LIN {X -0.004,Y -144.888,Z 390.932,A 0.000,B 0.000,C 90.000,E1 167.757} C_DIS
LIN {X -0.050,Y -147.516,Z 390.912,A 0.000,B 0.000,C 90.000,E1 164.102} C_DIS
LIN {X 0.025,Y -150.110,Z 390.891,A 0.000,B 0.000,C 90.000,E1 160.423} C_DIS
LIN {X 0.036,Y -153.470,Z 390.871,A 0.000,B 0.000,C 90.000,E1 156.794} C_DIS
LIN {X 0.027,Y -157.832,Z 390.846,A 0.000,B 0.000,C 90.000,E1 152.308} C_DIS
LIN {X 0.058,Y -162.117,Z 390.826,A 0.000,B 0.000,C 90.000,E1 148.742} C_DIS
LIN {X -0.057,Y -166.318,Z 390.807,A 0.000,B 0.000,C 90.000,E1 145.261} C_DIS
LIN {X 0.044,Y -171.337,Z 390.788,A 0.000,B 0.000,C 90.000,E1 141.743} C_DIS
LIN {X -0.027,Y -176.238,Z 390.768,A 0.000,B 0.000,C 90.000,E1 138.324} C_DIS
LIN {X 0.092,Y -180.518,Z 390.754,A 0.000,B 0.000,C 90.000,E1 135.729} C_DIS
LIN {X 0.072,Y -185.921,Z 390.736,A 0.000,B 0.000,C 90.000,E1 132.366} C_DIS
LIN {X 0.007,Y -190.550,Z 390.722,A 0.000,B 0.000,C 90.000,E1 129.886} C_DIS
LIN {X 0.038,Y -196.301,Z 390.703,A 0.000,B 0.000,C 90.000,E1 126.583} C_DIS
LIN {X -0.023,Y -198.087,Z 390.698,A 0.000,B 0.000,C 90.000,E1 125.678} C_DIS
LIN {X -0.088,Y -297.651,Z 390.698,A 0.000,B 0.000,C 90.000,E1 125.678} C_DIS
LIN {X -0.020,Y -298.876,Z 390.698,A 0.000,B 0.000,C 90.000,E1 125.644} C_DIS
LIN {X 0.001,Y -302.899,Z 390.697,A 0.000,B 0.000,C 90.000,E1 125.471} C_DIS
LIN {X -0.050,Y -305.154,Z 390.696,A 0.000,B 0.000,C 90.000,E1 125.311} C_DIS
LIN {X 0.098,Y -308.262,Z 390.694,A 0.000,B 0.000,C 90.000,E1 124.945} C_DIS
LIN {X 0.018,Y -310.260,Z 390.693,A 0.000,B 0.000,C 90.000,E1 124.659} C_DIS
LIN {X 0.019,Y -311.830,Z 390.691,A 0.000,B 0.000,C 90.000,E1 124.358} C_DIS
LIN {X -0.017,Y -313.176,Z 390.689,A 0.000,B 0.000,C 90.000,E1 124.040} C_DIS
LIN {X 0.147,Y -324.392,Z 390.671,A 0.000,B 0.000,C 90.000,E1 120.797} C_DIS
LIN {X 0.063,Y -335.861,Z 390.655,A 0.000,B 0.000,C 90.000,E1 117.975} C_DIS
LIN {X -0.012,Y -348.771,Z 390.640,A 0.000,B 0.000,C 90.000,E1 115.207} C_DIS
LIN {X 0.098,Y -361.555,Z 390.627,A 0.000,B 0.000,C 90.000,E1 112.770} C_DIS
LIN {X -0.081,Y -375.664,Z 390.613,A 0.000,B 0.000,C 90.000,E1 110.429} C_DIS
LIN {X -0.053,Y -391.204,Z 390.601,A 0.000,B 0.000,C 90.000,E1 108.109} C_DIS
LIN {X 0.000,Y -408.288,Z 390.588,A 0.000,B 0.000,C 90.000,E1 105.843} C_DIS
LIN {X -0.024,Y -427.043,Z 390.576,A 0.000,B 0.000,C 90.000,E1 103.647} C_DIS
LIN {X 0.196,Y -447.068,Z 390.564,A 0.000,B 0.000,C 90.000,E1 101.535} C_DIS
LIN {X -0.169,Y -467.667,Z 390.554,A 0.000,B 0.000,C 90.000,E1 99.670} C_DIS
LIN {X 0.207,Y -488.731,Z 390.544,A 0.000,B 0.000,C 90.000,E1 97.871} C_DIS
LIN {X -0.132,Y -490.860,Z 390.543,A 0.000,B 0.000,C 90.000,E1 97.701} C_DIS
LIN {X -0.189,Y -492.702,Z 390.541,A 0.000,B 0.000,C 90.000,E1 97.466} C_DIS
LIN {X 0.180,Y -494.092,Z 390.540,A 0.000,B 0.000,C 90.000,E1 97.182} C_DIS
LIN {X -0.070,Y -495.891,Z 390.537,A 0.000,B 0.000,C 90.000,E1 96.720} C_DIS
LIN {X 0.180,Y -496.581,Z 390.535,A 0.000,B 0.000,C 90.000,E1 96.201} C_DIS
LIN {X -0.053,Y -496.278,Z 390.532,A 0.000,B 0.000,C 90.000,E1 95.739} C_DIS
LIN {X 0.209,Y -494.934,Z 390.529,A 0.000,B 0.000,C 90.000,E1 95.220} C_DIS
LIN {X 0.070,Y -493.801,Z 390.528,A 0.000,B 0.000,C 90.000,E1 94.992} C_DIS
LIN {X -0.026,Y -492.278,Z 390.526,A 0.000,B 0.000,C 90.000,E1 94.759} C_DIS
LIN {X -0.088,Y -484.870,Z 390.521,A 0.000,B 0.000,C 90.000,E1 93.784} C_DIS
LIN {X 0.074,Y -474.923,Z 390.514,A 0.000,B 0.000,C 90.000,E1 92.522} C_DIS
LIN {X 0.199,Y -453.804,Z 390.499,A 0.000,B 0.000,C 90.000,E1 89.714} C_DIS
LIN {X 0.116,Y -434.527,Z 390.483,A 0.000,B 0.000,C 90.000,E1 86.849} C_DIS
LIN {X 0.076,Y -415.309,Z 390.465,A 0.000,B 0.000,C 90.000,E1 83.628} C_DIS
LIN {X -0.113,Y -406.122,Z 390.456,A 0.000,B 0.000,C 90.000,E1 82.008} C_DIS
LIN {X 0.166,Y -392.691,Z 390.442,A 0.000,B 0.000,C 90.000,E1 79.454} C_DIS
LIN {X 0.149,Y -382.343,Z 390.430,A 0.000,B 0.000,C 90.000,E1 77.465} C_DIS
LIN {X 0.002,Y -370.785,Z 390.418,A 0.000,B 0.000,C 90.000,E1 75.172} C_DIS
LIN {X -0.123,Y -359.363,Z 390.405,A 0.000,B 0.000,C 90.000,E1 72.834} C_DIS
LIN {X -0.031,Y -346.929,Z 390.389,A 0.000,B 0.000,C 90.000,E1 70.115} C_DIS
LIN {X -0.056,Y -334.832,Z 390.374,A 0.000,B 0.000,C 90.000,E1 67.358} C_DIS
LIN {X 0.010,Y -320.883,Z 390.355,A 0.000,B 0.000,C 90.000,E1 63.896} C_DIS
LIN {X -0.101,Y -307.827,Z 390.335,A 0.000,B 0.000,C 90.000,E1 60.383} C_DIS
LIN {X -0.017,Y -295.740,Z 390.315,A 0.000,B 0.000,C 90.000,E1 56.755} C_DIS
LIN {X -0.058,Y -285.753,Z 390.297,A 0.000,B 0.000,C 90.000,E1 53.417} C_DIS
LIN {X 0.025,Y -278.252,Z 390.282,A 0.000,B 0.000,C 90.000,E1 50.678} C_DIS
LIN {X 0.037,Y -272.653,Z 390.270,A 0.000,B 0.000,C 90.000,E1 48.609} C_DIS
LIN {X -0.050,Y -267.017,Z 390.258,A 0.000,B 0.000,C 90.000,E1 46.539} C_DIS
LIN {X -0.068,Y -261.180,Z 390.247,A 0.000,B 0.000,C 90.000,E1 44.433} C_DIS
LIN {X -0.010,Y -255.265,Z 390.235,A 0.000,B 0.000,C 90.000,E1 42.285} C_DIS
LIN {X 0.138,Y -249.210,Z 390.223,A 0.000,B 0.000,C 90.000,E1 40.092} C_DIS
LIN {X -0.141,Y -241.139,Z 390.207,A 0.000,B 0.000,C 90.000,E1 37.237} C_DIS
LIN {X -0.052,Y -231.567,Z 390.186,A 0.000,B 0.000,C 90.000,E1 33.499} C_DIS
LIN {X 0.119,Y -222.733,Z 390.165,A 0.000,B 0.000,C 90.000,E1 29.667} C_DIS
LIN {X 0.000,Y -216.307,Z 390.148,A 0.000,B 0.000,C 90.000,E1 26.616} C_DIS
LIN {X -0.038,Y -209.169,Z 390.126,A 0.000,B 0.000,C 90.000,E1 22.717} C_DIS
LIN {X 0.047,Y -203.101,Z 390.104,A 0.000,B 0.000,C 90.000,E1 18.725} C_DIS
LIN {X 0.004,Y -197.908,Z 390.082,A 0.000,B 0.000,C 90.000,E1 14.717} C_DIS
LIN {X -0.014,Y -193.670,Z 390.059,A 0.000,B 0.000,C 90.000,E1 10.658} C_DIS
LIN {X 0.015,Y -190.579,Z 390.036,A 0.000,B 0.000,C 90.000,E1 6.549} C_DIS
LIN {X 0.086,Y -188.349,Z 390.004,A 0.000,B 0.000,C 90.000,E1 0.745} C_DIS
LIN {X 0.094,Y -189.792,Z 389.947,A 0.000,B 0.000,C 90.000,E1 350.387} C_DIS
LIN {X 0.009,Y -192.664,Z 389.919,A 0.000,B 0.000,C 90.000,E1 345.463} C_DIS
LIN {X -0.115,Y -196.117,Z 389.896,A 0.000,B 0.000,C 90.000,E1 341.402} C_DIS
LIN {X -0.005,Y -200.733,Z 389.874,A 0.000,B 0.000,C 90.000,E1 337.305} C_DIS
LIN {X 0.097,Y -206.419,Z 389.852,A 0.000,B 0.000,C 90.000,E1 333.256} C_DIS
LIN {X -0.069,Y -213.025,Z 389.830,A 0.000,B 0.000,C 90.000,E1 329.331} C_DIS
LIN {X 0.040,Y -218.897,Z 389.812,A 0.000,B 0.000,C 90.000,E1 326.167} C_DIS
LIN {X -0.010,Y -226.615,Z 389.791,A 0.000,B 0.000,C 90.000,E1 322.316} C_DIS
LIN {X -0.063,Y -235.293,Z 389.770,A 0.000,B 0.000,C 90.000,E1 318.528} C_DIS
LIN {X -0.035,Y -244.257,Z 389.751,A 0.000,B 0.000,C 90.000,E1 315.162} C_DIS
LIN {X 0.101,Y -254.424,Z 389.733,A 0.000,B 0.000,C 90.000,E1 311.838} C_DIS
LIN {X 0.056,Y -265.861,Z 389.715,A 0.000,B 0.000,C 90.000,E1 308.624} C_DIS
LIN {X 0.124,Y -276.526,Z 389.699,A 0.000,B 0.000,C 90.000,E1 305.804} C_DIS
LIN {X -0.085,Y -290.732,Z 389.680,A 0.000,B 0.000,C 90.000,E1 302.418} C_DIS
LIN {X -0.109,Y -303.015,Z 389.665,A 0.000,B 0.000,C 90.000,E1 299.745} C_DIS
LIN {X -0.141,Y -320.332,Z 389.647,A 0.000,B 0.000,C 90.000,E1 296.488} C_DIS
LIN {X -0.074,Y -331.967,Z 389.636,A 0.000,B 0.000,C 90.000,E1 294.567} C_DIS
LIN {X -0.010,Y -353.439,Z 389.619,A 0.000,B 0.000,C 90.000,E1 291.461} C_DIS
LIN {X -0.073,Y -374.118,Z 389.604,A 0.000,B 0.000,C 90.000,E1 288.779} C_DIS
LIN {X 0.168,Y -391.598,Z 389.593,A 0.000,B 0.000,C 90.000,E1 286.732} C_DIS
LIN {X 0.151,Y -412.177,Z 389.581,A 0.000,B 0.000,C 90.000,E1 284.592} C_DIS
LIN {X -0.199,Y -425.093,Z 389.574,A 0.000,B 0.000,C 90.000,E1 283.355} C_DIS
LIN {X -0.020,Y -435.184,Z 389.568,A 0.000,B 0.000,C 90.000,E1 282.299} C_DIS
LIN {X 0.211,Y -442.512,Z 389.564,A 0.000,B 0.000,C 90.000,E1 281.478} C_DIS
LIN {X 0.124,Y -449.221,Z 389.560,A 0.000,B 0.000,C 90.000,E1 280.715} C_DIS
LIN {X -0.110,Y -455.551,Z 389.555,A 0.000,B 0.000,C 90.000,E1 279.962} C_DIS
LIN {X -0.015,Y -463.211,Z 389.550,A 0.000,B 0.000,C 90.000,E1 278.916} C_DIS
LIN {X 0.172,Y -470.157,Z 389.544,A 0.000,B 0.000,C 90.000,E1 277.871} C_DIS
LIN {X -0.093,Y -476.492,Z 389.538,A 0.000,B 0.000,C 90.000,E1 276.891} C_DIS
LIN {X -0.154,Y -480.751,Z 389.534,A 0.000,B 0.000,C 90.000,E1 276.144} C_DIS
LIN {X -0.125,Y -484.413,Z 389.530,A 0.000,B 0.000,C 90.000,E1 275.391} C_DIS
LIN {X 0.181,Y -485.505,Z 389.528,A 0.000,B 0.000,C 90.000,E1 275.106} C_DIS
LIN {X -0.116,Y -487.343,Z 389.526,A 0.000,B 0.000,C 90.000,E1 274.645} C_DIS
LIN {X 0.042,Y -488.781,Z 389.523,A 0.000,B 0.000,C 90.000,E1 274.131} C_DIS
LIN {X -0.242,Y -489.894,Z 389.520,A 0.000,B 0.000,C 90.000,E1 273.669} C_DIS
LIN {X -0.060,Y -490.710,Z 389.517,A 0.000,B 0.000,C 90.000,E1 273.154} C_DIS
LIN {X 0.156,Y -491.204,Z 389.515,A 0.000,B 0.000,C 90.000,E1 272.636} C_DIS
LIN {X -0.138,Y -491.394,Z 389.512,A 0.000,B 0.000,C 90.000,E1 272.178} C_DIS
LIN {X 0.079,Y -491.252,Z 389.509,A 0.000,B 0.000,C 90.000,E1 271.661} C_DIS
LIN {X -0.210,Y -490.728,Z 389.507,A 0.000,B 0.000,C 90.000,E1 271.203} C_DIS
LIN {X -0.008,Y -489.793,Z 389.504,A 0.000,B 0.000,C 90.000,E1 270.688} C_DIS
LIN {X 0.192,Y -488.460,Z 389.501,A 0.000,B 0.000,C 90.000,E1 270.172} C_DIS
LIN {X -0.102,Y -486.512,Z 389.498,A 0.000,B 0.000,C 90.000,E1 269.714} C_DIS
LIN {X 0.083,Y -483.942,Z 389.496,A 0.000,B 0.000,C 90.000,E1 269.198} C_DIS
LIN {X -0.076,Y -482.358,Z 389.494,A 0.000,B 0.000,C 90.000,E1 268.969} C_DIS
LIN {X 0.080,Y -478.442,Z 389.491,A 0.000,B 0.000,C 90.000,E1 268.453} C_DIS
LIN {X -0.086,Y -476.104,Z 389.490,A 0.000,B 0.000,C 90.000,E1 268.224} C_DIS
LIN {X 0.228,Y -473.451,Z 389.489,A 0.000,B 0.000,C 90.000,E1 267.936} C_DIS
LIN {X 0.052,Y -470.440,Z 389.487,A 0.000,B 0.000,C 90.000,E1 267.707} C_DIS
LIN {X 0.208,Y -464.101,Z 389.485,A 0.000,B 0.000,C 90.000,E1 267.249} C_DIS
LIN {X -0.021,Y -457.142,Z 389.483,A 0.000,B 0.000,C 90.000,E1 266.906} C_DIS
LIN {X -0.093,Y -449.997,Z 389.481,A 0.000,B 0.000,C 90.000,E1 266.617} C_DIS
LIN {X -0.179,Y -442.742,Z 389.480,A 0.000,B 0.000,C 90.000,E1 266.388} C_DIS
LIN {X 0.066,Y -434.559,Z 389.479,A 0.000,B 0.000,C 90.000,E1 266.159} C_DIS
LIN {X -0.089,Y -426.538,Z 389.478,A 0.000,B 0.000,C 90.000,E1 266.045} C_DIS
LIN {X 0.188,Y -419.861,Z 389.478,A 0.000,B 0.000,C 90.000,E1 265.931} C_DIS
LIN {X -0.075,Y -408.533,Z 389.477,A 0.000,B 0.000,C 90.000,E1 265.927} C_DIS
LIN {X -0.056,Y -180.917,Z 389.477,A 0.000,B 0.000,C 90.000,E1 265.927} C_DIS
LIN {X 0.067,Y -180.868,Z 389.472,A 0.000,B 0.000,C 90.000,E1 265.008} C_DIS
LIN {X -0.056,Y -178.984,Z 389.444,A 0.000,B 0.000,C 90.000,E1 259.982} C_DIS
LIN {X -0.044,Y -177.958,Z 389.435,A 0.000,B 0.000,C 90.000,E1 258.285} C_DIS
LIN {X -0.026,Y -175.599,Z 389.411,A 0.000,B 0.000,C 90.000,E1 254.031} C_DIS
LIN {X -0.013,Y -172.323,Z 389.387,A 0.000,B 0.000,C 90.000,E1 249.752} C_DIS
LIN {X -0.034,Y -171.801,Z 389.383,A 0.000,B 0.000,C 90.000,E1 248.901} C_DIS
LIN {X 0.004,Y -169.475,Z 389.368,A 0.000,B 0.000,C 90.000,E1 246.305} C_DIS
LIN {X -0.090,Y -166.802,Z 389.349,A 0.000,B 0.000,C 90.000,E1 242.871} C_DIS
LIN {X 0.053,Y -162.783,Z 389.325,A 0.000,B 0.000,C 90.000,E1 238.456} C_DIS
LIN {X 0.029,Y -161.471,Z 389.315,A 0.000,B 0.000,C 90.000,E1 236.707} C_DIS
LIN {X 0.070,Y -157.466,Z 389.291,A 0.000,B 0.000,C 90.000,E1 232.271} C_DIS
LIN {X 0.003,Y -155.480,Z 389.276,A 0.000,B 0.000,C 90.000,E1 229.622} C_DIS
LIN {X -0.065,Y -151.789,Z 389.251,A 0.000,B 0.000,C 90.000,E1 225.162} C_DIS
LIN {X -0.051,Y -149.997,Z 389.236,A 0.000,B 0.000,C 90.000,E1 222.447} C_DIS
LIN {X -0.019,Y -146.827,Z 389.210,A 0.000,B 0.000,C 90.000,E1 217.890} C_DIS
LIN {X -0.033,Y -145.407,Z 389.195,A 0.000,B 0.000,C 90.000,E1 215.152} C_DIS
LIN {X 0.003,Y -142.838,Z 389.170,A 0.000,B 0.000,C 90.000,E1 210.541} C_DIS
LIN {X -0.067,Y -141.451,Z 389.149,A 0.000,B 0.000,C 90.000,E1 206.873} C_DIS
LIN {X -0.027,Y -139.372,Z 389.113,A 0.000,B 0.000,C 90.000,E1 200.355} C_DIS
LIN {X -0.085,Y -138.821,Z 389.098,A 0.000,B 0.000,C 90.000,E1 197.583} C_DIS
LIN {X 0.004,Y -138.353,Z 389.056,A 0.000,B 0.000,C 90.000,E1 190.074} C_DIS
LIN {X -0.023,Y -139.533,Z 389.004,A 0.000,B 0.000,C 90.000,E1 180.745} C_DIS
LIN {X 0.070,Y -141.217,Z 388.973,A 0.000,B 0.000,C 90.000,E1 175.122} C_DIS
LIN {X 0.029,Y -142.591,Z 388.958,A 0.000,B 0.000,C 90.000,E1 172.356} C_DIS
LIN {X -0.017,Y -144.892,Z 388.932,A 0.000,B 0.000,C 90.000,E1 167.757} C_DIS
LIN {X -0.064,Y -147.519,Z 388.912,A 0.000,B 0.000,C 90.000,E1 164.102} C_DIS
LIN {X 0.010,Y -150.114,Z 388.891,A 0.000,B 0.000,C 90.000,E1 160.423} C_DIS
LIN {X 0.022,Y -153.475,Z 388.871,A 0.000,B 0.000,C 90.000,E1 156.794} C_DIS
LIN {X 0.086,Y -157.838,Z 388.846,A 0.000,B 0.000,C 90.000,E1 152.281} C_DIS
LIN {X 0.043,Y -162.123,Z 388.826,A 0.000,B 0.000,C 90.000,E1 148.742} C_DIS
LIN {X -0.072,Y -166.325,Z 388.807,A 0.000,B 0.000,C 90.000,E1 145.261} C_DIS
LIN {X 0.029,Y -171.343,Z 388.788,A 0.000,B 0.000,C 90.000,E1 141.743} C_DIS
LIN {X -0.044,Y -176.245,Z 388.768,A 0.000,B 0.000,C 90.000,E1 138.324} C_DIS
LIN {X 0.076,Y -180.527,Z 388.754,A 0.000,B 0.000,C 90.000,E1 135.729} C_DIS
LIN {X 0.056,Y -185.930,Z 388.735,A 0.000,B 0.000,C 90.000,E1 132.366} C_DIS
LIN {X -0.010,Y -190.560,Z 388.722,A 0.000,B 0.000,C 90.000,E1 129.886} C_DIS
LIN {X 0.021,Y -196.310,Z 388.703,A 0.000,B 0.000,C 90.000,E1 126.583} C_DIS
LIN {X 0.084,Y -198.184,Z 388.698,A 0.000,B 0.000,C 90.000,E1 125.598} C_DIS
LIN {X 0.090,Y -297.208,Z 388.698,A 0.000,B 0.000,C 90.000,E1 125.598} C_DIS
LIN {X -0.150,Y -299.822,Z 388.698,A 0.000,B 0.000,C 90.000,E1 125.598} C_DIS
LIN {X 0.173,Y -305.154,Z 388.696,A 0.000,B 0.000,C 90.000,E1 125.231} C_DIS
LIN {X 0.073,Y -308.048,Z 388.694,A 0.000,B 0.000,C 90.000,E1 124.945} C_DIS
LIN {X -0.144,Y -310.085,Z 388.693,A 0.000,B 0.000,C 90.000,E1 124.692} C_DIS
LIN {X -0.186,Y -311.685,Z 388.691,A 0.000,B 0.000,C 90.000,E1 124.405} C_DIS
LIN {X 0.037,Y -313.091,Z 388.689,A 0.000,B 0.000,C 90.000,E1 124.040} C_DIS
LIN {X 0.010,Y -325.542,Z 388.670,A 0.000,B 0.000,C 90.000,E1 120.512} C_DIS
LIN {X -0.052,Y -337.159,Z 388.654,A 0.000,B 0.000,C 90.000,E1 117.692} C_DIS
LIN {X 0.057,Y -350.234,Z 388.638,A 0.000,B 0.000,C 90.000,E1 114.899} C_DIS
LIN {X -0.126,Y -363.174,Z 388.625,A 0.000,B 0.000,C 90.000,E1 112.514} C_DIS
LIN {X 0.075,Y -377.452,Z 388.612,A 0.000,B 0.000,C 90.000,E1 110.120} C_DIS
LIN {X 0.030,Y -393.173,Z 388.599,A 0.000,B 0.000,C 90.000,E1 107.819} C_DIS
LIN {X 0.145,Y -410.453,Z 388.587,A 0.000,B 0.000,C 90.000,E1 105.552} C_DIS
LIN {X 0.187,Y -429.421,Z 388.574,A 0.000,B 0.000,C 90.000,E1 103.355} C_DIS
LIN {X 0.143,Y -449.531,Z 388.563,A 0.000,B 0.000,C 90.000,E1 101.299} C_DIS
LIN {X -0.144,Y -470.193,Z 388.552,A 0.000,B 0.000,C 90.000,E1 99.443} C_DIS
LIN {X 0.253,Y -488.647,Z 388.544,A 0.000,B 0.000,C 90.000,E1 97.871} C_DIS
LIN {X -0.087,Y -490.843,Z 388.543,A 0.000,B 0.000,C 90.000,E1 97.701} C_DIS
LIN {X -0.106,Y -492.706,Z 388.541,A 0.000,B 0.000,C 90.000,E1 97.466} C_DIS
LIN {X -0.189,Y -494.119,Z 388.540,A 0.000,B 0.000,C 90.000,E1 97.239} C_DIS
LIN {X 0.051,Y -495.999,Z 388.537,A 0.000,B 0.000,C 90.000,E1 96.720} C_DIS
LIN {X -0.192,Y -496.756,Z 388.535,A 0.000,B 0.000,C 90.000,E1 96.258} C_DIS
LIN {X 0.068,Y -496.516,Z 388.532,A 0.000,B 0.000,C 90.000,E1 95.739} C_DIS
LIN {X -0.162,Y -495.240,Z 388.529,A 0.000,B 0.000,C 90.000,E1 95.277} C_DIS
LIN {X 0.193,Y -494.151,Z 388.528,A 0.000,B 0.000,C 90.000,E1 94.992} C_DIS
LIN {X 0.097,Y -492.683,Z 388.526,A 0.000,B 0.000,C 90.000,E1 94.759} C_DIS
LIN {X 0.038,Y -485.314,Z 388.521,A 0.000,B 0.000,C 90.000,E1 93.784} C_DIS
LIN {X 0.029,Y -473.383,Z 388.513,A 0.000,B 0.000,C 90.000,E1 92.293} C_DIS
LIN {X 0.106,Y -452.367,Z 388.497,A 0.000,B 0.000,C 90.000,E1 89.484} C_DIS
LIN {X 0.011,Y -433.226,Z 388.481,A 0.000,B 0.000,C 90.000,E1 86.617} C_DIS
LIN {X -0.052,Y -414.135,Z 388.463,A 0.000,B 0.000,C 90.000,E1 83.394} C_DIS
LIN {X -0.107,Y -401.918,Z 388.451,A 0.000,B 0.000,C 90.000,E1 81.197} C_DIS
LIN {X 0.068,Y -390.103,Z 388.439,A 0.000,B 0.000,C 90.000,E1 78.926} C_DIS
LIN {X 0.028,Y -378.336,Z 388.426,A 0.000,B 0.000,C 90.000,E1 76.645} C_DIS
LIN {X -0.098,Y -369.692,Z 388.416,A 0.000,B 0.000,C 90.000,E1 74.921} C_DIS
LIN {X 0.002,Y -358.308,Z 388.403,A 0.000,B 0.000,C 90.000,E1 72.543} C_DIS
LIN {X 0.047,Y -345.870,Z 388.388,A 0.000,B 0.000,C 90.000,E1 69.826} C_DIS
LIN {X 0.109,Y -333.768,Z 388.373,A 0.000,B 0.000,C 90.000,E1 67.050} C_DIS
LIN {X -0.104,Y -321.088,Z 388.355,A 0.000,B 0.000,C 90.000,E1 63.948} C_DIS
LIN {X 0.072,Y -308.022,Z 388.336,A 0.000,B 0.000,C 90.000,E1 60.383} C_DIS
LIN {X 0.000,Y -295.936,Z 388.315,A 0.000,B 0.000,C 90.000,E1 56.786} C_DIS
LIN {X 0.121,Y -285.921,Z 388.297,A 0.000,B 0.000,C 90.000,E1 53.417} C_DIS
LIN {X -0.013,Y -278.431,Z 388.282,A 0.000,B 0.000,C 90.000,E1 50.723} C_DIS
LIN {X 0.035,Y -272.831,Z 388.270,A 0.000,B 0.000,C 90.000,E1 48.647} C_DIS
LIN {X 0.128,Y -267.200,Z 388.259,A 0.000,B 0.000,C 90.000,E1 46.539} C_DIS
LIN {X 0.109,Y -261.392,Z 388.247,A 0.000,B 0.000,C 90.000,E1 44.433} C_DIS
LIN {X -0.005,Y -255.491,Z 388.235,A 0.000,B 0.000,C 90.000,E1 42.324} C_DIS
LIN {X -0.037,Y -249.459,Z 388.223,A 0.000,B 0.000,C 90.000,E1 40.172} C_DIS
LIN {X 0.037,Y -241.383,Z 388.207,A 0.000,B 0.000,C 90.000,E1 37.237} C_DIS
LIN {X 0.126,Y -231.829,Z 388.186,A 0.000,B 0.000,C 90.000,E1 33.499} C_DIS
LIN {X -0.006,Y -222.957,Z 388.165,A 0.000,B 0.000,C 90.000,E1 29.745} C_DIS
LIN {X -0.016,Y -216.485,Z 388.148,A 0.000,B 0.000,C 90.000,E1 26.668} C_DIS
LIN {X -0.054,Y -209.291,Z 388.126,A 0.000,B 0.000,C 90.000,E1 22.770} C_DIS
LIN {X 0.031,Y -203.189,Z 388.104,A 0.000,B 0.000,C 90.000,E1 18.779} C_DIS
LIN {X -0.014,Y -197.946,Z 388.082,A 0.000,B 0.000,C 90.000,E1 14.773} C_DIS
LIN {X -0.033,Y -193.679,Z 388.059,A 0.000,B 0.000,C 90.000,E1 10.715} C_DIS
LIN {X -0.006,Y -190.532,Z 388.037,A 0.000,B 0.000,C 90.000,E1 6.606} C_DIS
LIN {X 0.062,Y -188.290,Z 388.005,A 0.000,B 0.000,C 90.000,E1 0.802} C_DIS
LIN {X 0.089,Y -189.686,Z 387.947,A 0.000,B 0.000,C 90.000,E1 350.387} C_DIS
LIN {X -0.001,Y -192.537,Z 387.919,A 0.000,B 0.000,C 90.000,E1 345.463} C_DIS
LIN {X 0.056,Y -195.990,Z 387.896,A 0.000,B 0.000,C 90.000,E1 341.348} C_DIS
LIN {X -0.023,Y -200.597,Z 387.874,A 0.000,B 0.000,C 90.000,E1 337.305} C_DIS
LIN {X 0.074,Y -206.283,Z 387.852,A 0.000,B 0.000,C 90.000,E1 333.256} C_DIS
LIN {X -0.097,Y -212.913,Z 387.829,A 0.000,B 0.000,C 90.000,E1 329.331} C_DIS
LIN {X 0.009,Y -218.781,Z 387.812,A 0.000,B 0.000,C 90.000,E1 326.167} C_DIS
LIN {X -0.046,Y -226.510,Z 387.791,A 0.000,B 0.000,C 90.000,E1 322.316} C_DIS
LIN {X 0.073,Y -235.179,Z 387.769,A 0.000,B 0.000,C 90.000,E1 318.485} C_DIS
LIN {X -0.080,Y -244.177,Z 387.751,A 0.000,B 0.000,C 90.000,E1 315.162} C_DIS
LIN {X 0.051,Y -254.349,Z 387.732,A 0.000,B 0.000,C 90.000,E1 311.838} C_DIS
LIN {X 0.002,Y -265.796,Z 387.715,A 0.000,B 0.000,C 90.000,E1 308.624} C_DIS
LIN {X 0.066,Y -276.464,Z 387.699,A 0.000,B 0.000,C 90.000,E1 305.804} C_DIS
LIN {X -0.149,Y -290.644,Z 387.680,A 0.000,B 0.000,C 90.000,E1 302.418} C_DIS
LIN {X -0.027,Y -302.998,Z 387.665,A 0.000,B 0.000,C 90.000,E1 299.716} C_DIS
LIN {X 0.150,Y -318.508,Z 387.649,A 0.000,B 0.000,C 90.000,E1 296.744} C_DIS
LIN {X 0.155,Y -332.048,Z 387.636,A 0.000,B 0.000,C 90.000,E1 294.515} C_DIS
LIN {X -0.111,Y -351.401,Z 387.621,A 0.000,B 0.000,C 90.000,E1 291.770} C_DIS
LIN {X -0.147,Y -374.340,Z 387.604,A 0.000,B 0.000,C 90.000,E1 288.779} C_DIS
LIN {X 0.145,Y -391.804,Z 387.593,A 0.000,B 0.000,C 90.000,E1 286.732} C_DIS
LIN {X 0.146,Y -412.364,Z 387.581,A 0.000,B 0.000,C 90.000,E1 284.592} C_DIS
LIN {X 0.127,Y -425.369,Z 387.574,A 0.000,B 0.000,C 90.000,E1 283.300} C_DIS
LIN {X -0.101,Y -435.481,Z 387.568,A 0.000,B 0.000,C 90.000,E1 282.299} C_DIS
LIN {X 0.164,Y -442.670,Z 387.564,A 0.000,B 0.000,C 90.000,E1 281.478} C_DIS
LIN {X -0.048,Y -449.436,Z 387.559,A 0.000,B 0.000,C 90.000,E1 280.715} C_DIS
LIN {X 0.167,Y -455.774,Z 387.555,A 0.000,B 0.000,C 90.000,E1 279.905} C_DIS
LIN {X -0.188,Y -463.358,Z 387.549,A 0.000,B 0.000,C 90.000,E1 278.916} C_DIS
LIN {X -0.001,Y -470.282,Z 387.544,A 0.000,B 0.000,C 90.000,E1 277.871} C_DIS
LIN {X -0.122,Y -475.087,Z 387.539,A 0.000,B 0.000,C 90.000,E1 277.125} C_DIS
LIN {X 0.148,Y -480.824,Z 387.534,A 0.000,B 0.000,C 90.000,E1 276.087} C_DIS
LIN {X 0.181,Y -484.464,Z 387.530,A 0.000,B 0.000,C 90.000,E1 275.334} C_DIS
LIN {X 0.193,Y -487.339,Z 387.526,A 0.000,B 0.000,C 90.000,E1 274.588} C_DIS
LIN {X -0.135,Y -488.825,Z 387.523,A 0.000,B 0.000,C 90.000,E1 274.131} C_DIS
LIN {X 0.069,Y -489.911,Z 387.520,A 0.000,B 0.000,C 90.000,E1 273.612} C_DIS
LIN {X -0.210,Y -490.706,Z 387.517,A 0.000,B 0.000,C 90.000,E1 273.151} C_DIS
LIN {X -0.021,Y -491.180,Z 387.515,A 0.000,B 0.000,C 90.000,E1 272.636} C_DIS
LIN {X 0.176,Y -491.364,Z 387.512,A 0.000,B 0.000,C 90.000,E1 272.121} C_DIS
LIN {X -0.098,Y -491.215,Z 387.509,A 0.000,B 0.000,C 90.000,E1 271.661} C_DIS
LIN {X 0.103,Y -490.686,Z 387.506,A 0.000,B 0.000,C 90.000,E1 271.146} C_DIS
LIN {X -0.185,Y -489.748,Z 387.504,A 0.000,B 0.000,C 90.000,E1 270.688} C_DIS
LIN {X 0.015,Y -488.387,Z 387.501,A 0.000,B 0.000,C 90.000,E1 270.172} C_DIS
LIN {X 0.208,Y -486.477,Z 387.498,A 0.000,B 0.000,C 90.000,E1 269.656} C_DIS
LIN {X -0.093,Y -483.888,Z 387.495,A 0.000,B 0.000,C 90.000,E1 269.198} C_DIS
LIN {X 0.072,Y -480.390,Z 387.493,A 0.000,B 0.000,C 90.000,E1 268.682} C_DIS
LIN {X -0.095,Y -478.376,Z 387.491,A 0.000,B 0.000,C 90.000,E1 268.453} C_DIS
LIN {X 0.054,Y -473.316,Z 387.489,A 0.000,B 0.000,C 90.000,E1 267.936} C_DIS
LIN {X -0.120,Y -470.315,Z 387.487,A 0.000,B 0.000,C 90.000,E1 267.707} C_DIS
LIN {X -0.045,Y -467.301,Z 387.486,A 0.000,B 0.000,C 90.000,E1 267.478} C_DIS
LIN {X -0.056,Y -460.651,Z 387.484,A 0.000,B 0.000,C 90.000,E1 267.078} C_DIS
LIN {X 0.064,Y -453.637,Z 387.482,A 0.000,B 0.000,C 90.000,E1 266.731} C_DIS
LIN {X 0.203,Y -446.421,Z 387.480,A 0.000,B 0.000,C 90.000,E1 266.445} C_DIS
LIN {X -0.131,Y -439.021,Z 387.479,A 0.000,B 0.000,C 90.000,E1 266.274} C_DIS
LIN {X -0.071,Y -430.842,Z 387.478,A 0.000,B 0.000,C 90.000,E1 266.102} C_DIS
LIN {X 0.136,Y -419.623,Z 387.478,A 0.000,B 0.000,C 90.000,E1 265.931} C_DIS
LIN {X -0.070,Y -412.711,Z 387.477,A 0.000,B 0.000,C 90.000,E1 265.927} C_DIS
LIN {X -0.053,Y -180.917,Z 387.477,A 0.000,B 0.000,C 90.000,E1 265.927} C_DIS
LIN {X 0.049,Y -180.867,Z 387.472,A 0.000,B 0.000,C 90.000,E1 265.008} C_DIS
LIN {X -0.074,Y -178.982,Z 387.444,A 0.000,B 0.000,C 90.000,E1 259.982} C_DIS
LIN {X -0.062,Y -177.953,Z 387.435,A 0.000,B 0.000,C 90.000,E1 258.285} C_DIS
LIN {X -0.043,Y -175.595,Z 387.411,A 0.000,B 0.000,C 90.000,E1 254.031} C_DIS
LIN {X -0.030,Y -172.320,Z 387.387,A 0.000,B 0.000,C 90.000,E1 249.752} C_DIS
LIN {X -0.051,Y -171.797,Z 387.383,A 0.000,B 0.000,C 90.000,E1 248.901} C_DIS
LIN {X -0.014,Y -169.469,Z 387.368,A 0.000,B 0.000,C 90.000,E1 246.305} C_DIS
LIN {X 0.042,Y -166.797,Z 387.349,A 0.000,B 0.000,C 90.000,E1 242.820} C_DIS
LIN {X 0.036,Y -162.778,Z 387.325,A 0.000,B 0.000,C 90.000,E1 238.456} C_DIS
LIN {X 0.012,Y -161.467,Z 387.315,A 0.000,B 0.000,C 90.000,E1 236.707} C_DIS
LIN {X 0.053,Y -157.461,Z 387.290,A 0.000,B 0.000,C 90.000,E1 232.271} C_DIS
LIN {X -0.014,Y -155.473,Z 387.276,A 0.000,B 0.000,C 90.000,E1 229.622} C_DIS
LIN {X -0.081,Y -151.784,Z 387.251,A 0.000,B 0.000,C 90.000,E1 225.162} C_DIS
LIN {X -0.068,Y -149.992,Z 387.236,A 0.000,B 0.000,C 90.000,E1 222.447} C_DIS
LIN {X -0.035,Y -146.823,Z 387.210,A 0.000,B 0.000,C 90.000,E1 217.890} C_DIS
LIN {X 0.070,Y -145.402,Z 387.195,A 0.000,B 0.000,C 90.000,E1 215.105} C_DIS
LIN {X -0.013,Y -142.835,Z 387.170,A 0.000,B 0.000,C 90.000,E1 210.541} C_DIS
LIN {X 0.044,Y -141.448,Z 387.149,A 0.000,B 0.000,C 90.000,E1 206.821} C_DIS
LIN {X -0.043,Y -139.371,Z 387.113,A 0.000,B 0.000,C 90.000,E1 200.355} C_DIS
LIN {X 0.032,Y -138.819,Z 387.097,A 0.000,B 0.000,C 90.000,E1 197.528} C_DIS
LIN {X -0.012,Y -138.352,Z 387.056,A 0.000,B 0.000,C 90.000,E1 190.074} C_DIS
LIN {X -0.039,Y -139.534,Z 387.004,A 0.000,B 0.000,C 90.000,E1 180.745} C_DIS
LIN {X 0.054,Y -141.220,Z 386.973,A 0.000,B 0.000,C 90.000,E1 175.122} C_DIS
LIN {X 0.013,Y -142.593,Z 386.958,A 0.000,B 0.000,C 90.000,E1 172.356} C_DIS
LIN {X -0.034,Y -144.895,Z 386.932,A 0.000,B 0.000,C 90.000,E1 167.757} C_DIS
LIN {X -0.080,Y -147.524,Z 386.911,A 0.000,B 0.000,C 90.000,E1 164.102} C_DIS
LIN {X -0.006,Y -150.120,Z 386.891,A 0.000,B 0.000,C 90.000,E1 160.423} C_DIS
LIN {X 0.005,Y -153.482,Z 386.871,A 0.000,B 0.000,C 90.000,E1 156.794} C_DIS
LIN {X 0.069,Y -157.845,Z 386.846,A 0.000,B 0.000,C 90.000,E1 152.281} C_DIS
LIN {X 0.025,Y -162.131,Z 386.826,A 0.000,B 0.000,C 90.000,E1 148.742} C_DIS
LIN {X 0.005,Y -166.333,Z 386.807,A 0.000,B 0.000,C 90.000,E1 145.229} C_DIS
LIN {X 0.011,Y -171.351,Z 386.787,A 0.000,B 0.000,C 90.000,E1 141.743} C_DIS
LIN {X -0.062,Y -176.255,Z 386.768,A 0.000,B 0.000,C 90.000,E1 138.324} C_DIS
LIN {X 0.057,Y -180.538,Z 386.754,A 0.000,B 0.000,C 90.000,E1 135.729} C_DIS
LIN {X 0.037,Y -185.939,Z 386.735,A 0.000,B 0.000,C 90.000,E1 132.366} C_DIS
LIN {X -0.029,Y -190.570,Z 386.722,A 0.000,B 0.000,C 90.000,E1 129.886} C_DIS
LIN {X 0.002,Y -196.320,Z 386.703,A 0.000,B 0.000,C 90.000,E1 126.583} C_DIS
LIN {X -0.086,Y -198.281,Z 386.698,A 0.000,B 0.000,C 90.000,E1 125.598} C_DIS
LIN {X -0.180,Y -297.492,Z 386.698,A 0.000,B 0.000,C 90.000,E1 125.598} C_DIS
LIN {X 0.102,Y -302.486,Z 386.697,A 0.000,B 0.000,C 90.000,E1 125.391} C_DIS
LIN {X 0.142,Y -304.752,Z 386.696,A 0.000,B 0.000,C 90.000,E1 125.231} C_DIS
LIN {X 0.042,Y -307.824,Z 386.694,A 0.000,B 0.000,C 90.000,E1 124.945} C_DIS
LIN {X -0.073,Y -311.471,Z 386.691,A 0.000,B 0.000,C 90.000,E1 124.405} C_DIS
LIN {X -0.033,Y -312.959,Z 386.689,A 0.000,B 0.000,C 90.000,E1 124.072} C_DIS
LIN {X -0.055,Y -325.454,Z 386.670,A 0.000,B 0.000,C 90.000,E1 120.541} C_DIS
LIN {X -0.109,Y -337.061,Z 386.654,A 0.000,B 0.000,C 90.000,E1 117.719} C_DIS
LIN {X 0.158,Y -350.128,Z 386.638,A 0.000,B 0.000,C 90.000,E1 114.899} C_DIS
LIN {X -0.024,Y -363.058,Z 386.625,A 0.000,B 0.000,C 90.000,E1 112.514} C_DIS
LIN {X 0.178,Y -377.326,Z 386.612,A 0.000,B 0.000,C 90.000,E1 110.120} C_DIS
LIN {X 0.135,Y -393.037,Z 386.599,A 0.000,B 0.000,C 90.000,E1 107.819} C_DIS
LIN {X -0.144,Y -410.306,Z 386.587,A 0.000,B 0.000,C 90.000,E1 105.607} C_DIS
LIN {X -0.124,Y -429.262,Z 386.574,A 0.000,B 0.000,C 90.000,E1 103.411} C_DIS
LIN {X 0.245,Y -449.367,Z 386.563,A 0.000,B 0.000,C 90.000,E1 101.299} C_DIS
LIN {X -0.047,Y -470.025,Z 386.552,A 0.000,B 0.000,C 90.000,E1 99.443} C_DIS
LIN {X -0.205,Y -488.485,Z 386.544,A 0.000,B 0.000,C 90.000,E1 97.936} C_DIS
LIN {X 0.006,Y -490.774,Z 386.543,A 0.000,B 0.000,C 90.000,E1 97.701} C_DIS
LIN {X 0.036,Y -492.661,Z 386.542,A 0.000,B 0.000,C 90.000,E1 97.466} C_DIS
LIN {X 0.002,Y -494.100,Z 386.540,A 0.000,B 0.000,C 90.000,E1 97.239} C_DIS
LIN {X -0.250,Y -496.084,Z 386.537,A 0.000,B 0.000,C 90.000,E1 96.777} C_DIS
LIN {X 0.000,Y -496.923,Z 386.535,A 0.000,B 0.000,C 90.000,E1 96.258} C_DIS
LIN {X -0.233,Y -496.758,Z 386.532,A 0.000,B 0.000,C 90.000,E1 95.796} C_DIS
LIN {X 0.031,Y -495.569,Z 386.529,A 0.000,B 0.000,C 90.000,E1 95.277} C_DIS
LIN {X -0.106,Y -494.531,Z 386.528,A 0.000,B 0.000,C 90.000,E1 95.049} C_DIS
LIN {X -0.200,Y -493.127,Z 386.527,A 0.000,B 0.000,C 90.000,E1 94.816} C_DIS
LIN {X -0.139,Y -487.701,Z 386.523,A 0.000,B 0.000,C 90.000,E1 94.073} C_DIS
LIN {X -0.214,Y -479.903,Z 386.517,A 0.000,B 0.000,C 90.000,E1 93.094} C_DIS
LIN {X 0.087,Y -454.686,Z 386.499,A 0.000,B 0.000,C 90.000,E1 89.771} C_DIS
LIN {X 0.036,Y -435.315,Z 386.483,A 0.000,B 0.000,C 90.000,E1 86.906} C_DIS
LIN {X 0.027,Y -416.034,Z 386.465,A 0.000,B 0.000,C 90.000,E1 83.685} C_DIS
LIN {X -0.093,Y -405.337,Z 386.454,A 0.000,B 0.000,C 90.000,E1 81.781} C_DIS
LIN {X 0.224,Y -391.988,Z 386.440,A 0.000,B 0.000,C 90.000,E1 79.218} C_DIS
LIN {X 0.197,Y -381.653,Z 386.429,A 0.000,B 0.000,C 90.000,E1 77.229} C_DIS
LIN {X 0.034,Y -371.547,Z 386.418,A 0.000,B 0.000,C 90.000,E1 75.227} C_DIS
LIN {X -0.177,Y -360.109,Z 386.405,A 0.000,B 0.000,C 90.000,E1 72.906} C_DIS
LIN {X -0.108,Y -348.952,Z 386.392,A 0.000,B 0.000,C 90.000,E1 70.496} C_DIS
LIN {X 0.043,Y -338.068,Z 386.378,A 0.000,B 0.000,C 90.000,E1 68.028} C_DIS
LIN {X -0.012,Y -325.069,Z 386.361,A 0.000,B 0.000,C 90.000,E1 64.921} C_DIS
LIN {X 0.141,Y -311.710,Z 386.341,A 0.000,B 0.000,C 90.000,E1 61.385} C_DIS
LIN {X 0.150,Y -300.413,Z 386.323,A 0.000,B 0.000,C 90.000,E1 58.122} C_DIS
LIN {X 0.083,Y -290.048,Z 386.305,A 0.000,B 0.000,C 90.000,E1 54.815} C_DIS
LIN {X -0.030,Y -280.480,Z 386.286,A 0.000,B 0.000,C 90.000,E1 51.457} C_DIS
LIN {X 0.061,Y -274.933,Z 386.274,A 0.000,B 0.000,C 90.000,E1 49.380} C_DIS
LIN {X -0.023,Y -267.417,Z 386.259,A 0.000,B 0.000,C 90.000,E1 46.620} C_DIS
LIN {X -0.035,Y -261.634,Z 386.247,A 0.000,B 0.000,C 90.000,E1 44.514} C_DIS
LIN {X 0.031,Y -255.757,Z 386.235,A 0.000,B 0.000,C 90.000,E1 42.366} C_DIS
LIN {X -0.004,Y -249.736,Z 386.223,A 0.000,B 0.000,C 90.000,E1 40.216} C_DIS
LIN {X -0.078,Y -241.644,Z 386.207,A 0.000,B 0.000,C 90.000,E1 37.317} C_DIS
LIN {X 0.027,Y -232.104,Z 386.187,A 0.000,B 0.000,C 90.000,E1 33.579} C_DIS
LIN {X 0.023,Y -223.211,Z 386.166,A 0.000,B 0.000,C 90.000,E1 29.795} C_DIS
LIN {X -0.084,Y -216.688,Z 386.148,A 0.000,B 0.000,C 90.000,E1 26.744} C_DIS
LIN {X -0.026,Y -209.433,Z 386.127,A 0.000,B 0.000,C 90.000,E1 22.823} C_DIS
LIN {X -0.009,Y -203.295,Z 386.105,A 0.000,B 0.000,C 90.000,E1 18.852} C_DIS
LIN {X 0.011,Y -198.005,Z 386.082,A 0.000,B 0.000,C 90.000,E1 14.828} C_DIS
LIN {X -0.046,Y -193.703,Z 386.060,A 0.000,B 0.000,C 90.000,E1 10.782} C_DIS
LIN {X 0.015,Y -190.523,Z 386.037,A 0.000,B 0.000,C 90.000,E1 6.663} C_DIS
LIN {X 0.081,Y -188.245,Z 386.005,A 0.000,B 0.000,C 90.000,E1 0.859} C_DIS
LIN {X 0.084,Y -189.578,Z 385.947,A 0.000,B 0.000,C 90.000,E1 350.387} C_DIS
LIN {X -0.009,Y -192.409,Z 385.919,A 0.000,B 0.000,C 90.000,E1 345.463} C_DIS
LIN {X 0.044,Y -195.869,Z 385.896,A 0.000,B 0.000,C 90.000,E1 341.348} C_DIS
LIN {X 0.037,Y -200.458,Z 385.874,A 0.000,B 0.000,C 90.000,E1 337.283} C_DIS
LIN {X 0.053,Y -206.173,Z 385.852,A 0.000,B 0.000,C 90.000,E1 333.256} C_DIS
LIN {X 0.060,Y -212.818,Z 385.829,A 0.000,B 0.000,C 90.000,E1 329.282} C_DIS
LIN {X -0.021,Y -218.652,Z 385.812,A 0.000,B 0.000,C 90.000,E1 326.167} C_DIS
LIN {X 0.099,Y -226.408,Z 385.791,A 0.000,B 0.000,C 90.000,E1 322.271} C_DIS
LIN {X 0.033,Y -235.070,Z 385.769,A 0.000,B 0.000,C 90.000,E1 318.485} C_DIS
LIN {X -0.123,Y -244.100,Z 385.751,A 0.000,B 0.000,C 90.000,E1 315.162} C_DIS
LIN {X 0.004,Y -254.271,Z 385.732,A 0.000,B 0.000,C 90.000,E1 311.838} C_DIS
LIN {X -0.049,Y -265.719,Z 385.715,A 0.000,B 0.000,C 90.000,E1 308.624} C_DIS
LIN {X 0.010,Y -276.396,Z 385.699,A 0.000,B 0.000,C 90.000,E1 305.804} C_DIS
LIN {X 0.191,Y -290.567,Z 385.680,A 0.000,B 0.000,C 90.000,E1 302.339} C_DIS
LIN {X 0.171,Y -302.975,Z 385.665,A 0.000,B 0.000,C 90.000,E1 299.667} C_DIS
LIN {X 0.081,Y -318.541,Z 385.649,A 0.000,B 0.000,C 90.000,E1 296.744} C_DIS
LIN {X -0.017,Y -330.117,Z 385.638,A 0.000,B 0.000,C 90.000,E1 294.847} C_DIS
LIN {X 0.128,Y -349.373,Z 385.622,A 0.000,B 0.000,C 90.000,E1 292.025} C_DIS
LIN {X 0.088,Y -369.782,Z 385.607,A 0.000,B 0.000,C 90.000,E1 289.322} C_DIS
LIN {X 0.108,Y -387.058,Z 385.596,A 0.000,B 0.000,C 90.000,E1 287.275} C_DIS
LIN {X -0.149,Y -407.642,Z 385.584,A 0.000,B 0.000,C 90.000,E1 285.134} C_DIS
LIN {X 0.030,Y -423.300,Z 385.575,A 0.000,B 0.000,C 90.000,E1 283.536} C_DIS
LIN {X -0.198,Y -433.472,Z 385.569,A 0.000,B 0.000,C 90.000,E1 282.535} C_DIS
LIN {X 0.041,Y -440.802,Z 385.565,A 0.000,B 0.000,C 90.000,E1 281.715} C_DIS
LIN {X -0.179,Y -447.695,Z 385.561,A 0.000,B 0.000,C 90.000,E1 280.950} C_DIS
LIN {X -0.179,Y -456.112,Z 385.555,A 0.000,B 0.000,C 90.000,E1 279.905} C_DIS
LIN {X 0.096,Y -461.845,Z 385.551,A 0.000,B 0.000,C 90.000,E1 279.095} C_DIS
LIN {X -0.192,Y -468.873,Z 385.545,A 0.000,B 0.000,C 90.000,E1 278.106} C_DIS
LIN {X -0.001,Y -475.303,Z 385.539,A 0.000,B 0.000,C 90.000,E1 277.068} C_DIS
LIN {X -0.203,Y -481.005,Z 385.534,A 0.000,B 0.000,C 90.000,E1 276.087} C_DIS
LIN {X -0.172,Y -484.618,Z 385.530,A 0.000,B 0.000,C 90.000,E1 275.334} C_DIS
LIN {X -0.160,Y -487.442,Z 385.525,A 0.000,B 0.000,C 90.000,E1 274.588} C_DIS
LIN {X -0.001,Y -488.873,Z 385.523,A 0.000,B 0.000,C 90.000,E1 274.073} C_DIS
LIN {X 0.205,Y -489.942,Z 385.520,A 0.000,B 0.000,C 90.000,E1 273.555} C_DIS
LIN {X -0.075,Y -490.716,Z 385.517,A 0.000,B 0.000,C 90.000,E1 273.094} C_DIS
LIN {X 0.114,Y -491.177,Z 385.514,A 0.000,B 0.000,C 90.000,E1 272.579} C_DIS
LIN {X -0.179,Y -491.319,Z 385.512,A 0.000,B 0.000,C 90.000,E1 272.121} C_DIS
LIN {X 0.038,Y -491.130,Z 385.509,A 0.000,B 0.000,C 90.000,E1 271.604} C_DIS
LIN {X 0.239,Y -490.597,Z 385.506,A 0.000,B 0.000,C 90.000,E1 271.088} C_DIS
LIN {X -0.049,Y -489.654,Z 385.503,A 0.000,B 0.000,C 90.000,E1 270.630} C_DIS
LIN {X 0.149,Y -488.258,Z 385.501,A 0.000,B 0.000,C 90.000,E1 270.115} C_DIS
LIN {X -0.145,Y -486.264,Z 385.498,A 0.000,B 0.000,C 90.000,E1 269.656} C_DIS
LIN {X 0.039,Y -483.683,Z 385.495,A 0.000,B 0.000,C 90.000,E1 269.141} C_DIS
LIN {X 0.201,Y -480.192,Z 385.492,A 0.000,B 0.000,C 90.000,E1 268.625} C_DIS
LIN {X -0.118,Y -475.695,Z 385.490,A 0.000,B 0.000,C 90.000,E1 268.165} C_DIS
LIN {X 0.181,Y -472.997,Z 385.488,A 0.000,B 0.000,C 90.000,E1 267.879} C_DIS
LIN {X 0.004,Y -469.921,Z 385.487,A 0.000,B 0.000,C 90.000,E1 267.650} C_DIS
LIN {X 0.107,Y -466.938,Z 385.486,A 0.000,B 0.000,C 90.000,E1 267.421} C_DIS
LIN {X 0.160,Y -460.245,Z 385.484,A 0.000,B 0.000,C 90.000,E1 267.020} C_DIS
LIN {X 0.111,Y -456.725,Z 385.483,A 0.000,B 0.000,C 90.000,E1 266.849} C_DIS
LIN {X 0.032,Y -449.289,Z 385.481,A 0.000,B 0.000,C 90.000,E1 266.560} C_DIS
LIN {X -0.011,Y -441.961,Z 385.480,A 0.000,B 0.000,C 90.000,E1 266.331} C_DIS
LIN {X -0.104,Y -434.172,Z 385.479,A 0.000,B 0.000,C 90.000,E1 266.159} C_DIS
LIN {X 0.174,Y -425.900,Z 385.478,A 0.000,B 0.000,C 90.000,E1 265.988} C_DIS
LIN {X 0.068,Y -418.557,Z 385.477,A 0.000,B 0.000,C 90.000,E1 265.927} C_DIS
LIN {X -0.114,Y -412.308,Z 385.477,A 0.000,B 0.000,C 90.000,E1 265.927} C_DIS
LIN {X -0.071,Y -180.916,Z 385.477,A 0.000,B 0.000,C 90.000,E1 265.927} C_DIS
LIN {X 0.023,Y -180.865,Z 385.472,A 0.000,B 0.000,C 90.000,E1 265.008} C_DIS
LIN {X 0.075,Y -178.979,Z 385.444,A 0.000,B 0.000,C 90.000,E1 259.926} C_DIS
LIN {X 0.085,Y -177.948,Z 385.435,A 0.000,B 0.000,C 90.000,E1 258.229} C_DIS
LIN {X -0.069,Y -175.589,Z 385.411,A 0.000,B 0.000,C 90.000,E1 254.031} C_DIS
LIN {X -0.056,Y -172.314,Z 385.387,A 0.000,B 0.000,C 90.000,E1 249.752} C_DIS
LIN {X -0.077,Y -171.792,Z 385.383,A 0.000,B 0.000,C 90.000,E1 248.901} C_DIS
LIN {X -0.039,Y -169.462,Z 385.368,A 0.000,B 0.000,C 90.000,E1 246.305} C_DIS
LIN {X 0.016,Y -166.791,Z 385.349,A 0.000,B 0.000,C 90.000,E1 242.820} C_DIS
LIN {X 0.012,Y -162.770,Z 385.325,A 0.000,B 0.000,C 90.000,E1 238.456} C_DIS
LIN {X -0.012,Y -161.460,Z 385.315,A 0.000,B 0.000,C 90.000,E1 236.707} C_DIS
LIN {X 0.029,Y -157.454,Z 385.290,A 0.000,B 0.000,C 90.000,E1 232.271} C_DIS
LIN {X -0.038,Y -155.465,Z 385.276,A 0.000,B 0.000,C 90.000,E1 229.622} C_DIS
LIN {X 0.003,Y -151.779,Z 385.251,A 0.000,B 0.000,C 90.000,E1 225.121} C_DIS
LIN {X 0.020,Y -149.985,Z 385.236,A 0.000,B 0.000,C 90.000,E1 222.405} C_DIS
LIN {X -0.059,Y -146.817,Z 385.210,A 0.000,B 0.000,C 90.000,E1 217.890} C_DIS
LIN {X 0.047,Y -145.396,Z 385.195,A 0.000,B 0.000,C 90.000,E1 215.105} C_DIS
LIN {X -0.035,Y -142.831,Z 385.170,A 0.000,B 0.000,C 90.000,E1 210.541} C_DIS
LIN {X 0.021,Y -141.444,Z 385.149,A 0.000,B 0.000,C 90.000,E1 206.821} C_DIS
LIN {X 0.065,Y -139.369,Z 385.113,A 0.000,B 0.000,C 90.000,E1 200.301} C_DIS
LIN {X 0.051,Y -138.817,Z 385.097,A 0.000,B 0.000,C 90.000,E1 197.511} C_DIS
LIN {X -0.034,Y -138.352,Z 385.056,A 0.000,B 0.000,C 90.000,E1 190.074} C_DIS
LIN {X -0.061,Y -139.536,Z 385.004,A 0.000,B 0.000,C 90.000,E1 180.745} C_DIS
LIN {X 0.032,Y -141.225,Z 384.973,A 0.000,B 0.000,C 90.000,E1 175.122} C_DIS
LIN {X -0.010,Y -142.596,Z 384.958,A 0.000,B 0.000,C 90.000,E1 172.356} C_DIS
LIN {X -0.056,Y -144.901,Z 384.932,A 0.000,B 0.000,C 90.000,E1 167.757} C_DIS
LIN {X 0.038,Y -147.529,Z 384.911,A 0.000,B 0.000,C 90.000,E1 164.047} C_DIS
LIN {X -0.030,Y -150.127,Z 384.891,A 0.000,B 0.000,C 90.000,E1 160.423} C_DIS
LIN {X -0.018,Y -153.491,Z 384.871,A 0.000,B 0.000,C 90.000,E1 156.794} C_DIS
LIN {X 0.045,Y -157.855,Z 384.846,A 0.000,B 0.000,C 90.000,E1 152.281} C_DIS
LIN {X 0.001,Y -162.141,Z 384.826,A 0.000,B 0.000,C 90.000,E1 148.742} C_DIS
LIN {X -0.021,Y -166.345,Z 384.807,A 0.000,B 0.000,C 90.000,E1 145.229} C_DIS
LIN {X -0.015,Y -171.362,Z 384.787,A 0.000,B 0.000,C 90.000,E1 141.743} C_DIS
LIN {X -0.087,Y -176.268,Z 384.768,A 0.000,B 0.000,C 90.000,E1 138.324} C_DIS
LIN {X 0.031,Y -180.552,Z 384.754,A 0.000,B 0.000,C 90.000,E1 135.729} C_DIS
LIN {X 0.010,Y -185.954,Z 384.735,A 0.000,B 0.000,C 90.000,E1 132.366} C_DIS
LIN {X 0.066,Y -190.586,Z 384.721,A 0.000,B 0.000,C 90.000,E1 129.850} C_DIS
LIN {X -0.027,Y -196.335,Z 384.703,A 0.000,B 0.000,C 90.000,E1 126.583} C_DIS
LIN {X 0.000,Y -198.390,Z 384.697,A 0.000,B 0.000,C 90.000,E1 125.518} C_DIS
LIN {X -0.049,Y -298.045,Z 384.697,A 0.000,B 0.000,C 90.000,E1 125.518} C_DIS
LIN {X -0.149,Y -299.228,Z 384.697,A 0.000,B 0.000,C 90.000,E1 125.518} C_DIS
LIN {X -0.076,Y -304.767,Z 384.696,A 0.000,B 0.000,C 90.000,E1 125.231} C_DIS
LIN {X -0.001,Y -307.604,Z 384.694,A 0.000,B 0.000,C 90.000,E1 124.945} C_DIS
LIN {X -0.036,Y -311.313,Z 384.691,A 0.000,B 0.000,C 90.000,E1 124.405} C_DIS
LIN {X 0.003,Y -312.866,Z 384.689,A 0.000,B 0.000,C 90.000,E1 124.072} C_DIS
LIN {X 0.070,Y -316.228,Z 384.684,A 0.000,B 0.000,C 90.000,E1 123.086} C_DIS
LIN {X 0.078,Y -326.629,Z 384.668,A 0.000,B 0.000,C 90.000,E1 120.207} C_DIS
LIN {X 0.055,Y -338.392,Z 384.652,A 0.000,B 0.000,C 90.000,E1 117.385} C_DIS
LIN {X -0.101,Y -351.620,Z 384.637,A 0.000,B 0.000,C 90.000,E1 114.643} C_DIS
LIN {X 0.079,Y -364.709,Z 384.623,A 0.000,B 0.000,C 90.000,E1 112.206} C_DIS
LIN {X -0.029,Y -379.147,Z 384.610,A 0.000,B 0.000,C 90.000,E1 109.866} C_DIS
LIN {X -0.163,Y -395.042,Z 384.598,A 0.000,B 0.000,C 90.000,E1 107.583} C_DIS
LIN {X -0.005,Y -412.510,Z 384.585,A 0.000,B 0.000,C 90.000,E1 105.315} C_DIS
LIN {X 0.100,Y -431.658,Z 384.573,A 0.000,B 0.000,C 90.000,E1 103.119} C_DIS
LIN {X 0.124,Y -451.835,Z 384.562,A 0.000,B 0.000,C 90.000,E1 101.074} C_DIS
LIN {X 0.077,Y -472.556,Z 384.551,A 0.000,B 0.000,C 90.000,E1 99.208} C_DIS
LIN {X -0.176,Y -488.412,Z 384.544,A 0.000,B 0.000,C 90.000,E1 97.936} C_DIS
LIN {X 0.034,Y -490.765,Z 384.543,A 0.000,B 0.000,C 90.000,E1 97.701} C_DIS
LIN {X 0.034,Y -492.671,Z 384.542,A 0.000,B 0.000,C 90.000,E1 97.473} C_DIS
LIN {X 0.099,Y -494.126,Z 384.540,A 0.000,B 0.000,C 90.000,E1 97.239} C_DIS
LIN {X 0.005,Y -495.316,Z 384.539,A 0.000,B 0.000,C 90.000,E1 97.004} C_DIS
LIN {X -0.152,Y -496.180,Z 384.538,A 0.000,B 0.000,C 90.000,E1 96.777} C_DIS
LIN {X 0.105,Y -497.072,Z 384.535,A 0.000,B 0.000,C 90.000,E1 96.258} C_DIS
LIN {X -0.128,Y -496.967,Z 384.532,A 0.000,B 0.000,C 90.000,E1 95.796} C_DIS
LIN {X 0.137,Y -495.840,Z 384.529,A 0.000,B 0.000,C 90.000,E1 95.277} C_DIS
LIN {X 0.000,Y -494.841,Z 384.528,A 0.000,B 0.000,C 90.000,E1 95.049} C_DIS
LIN {X -0.135,Y -493.483,Z 384.527,A 0.000,B 0.000,C 90.000,E1 94.821} C_DIS
LIN {X -0.031,Y -488.133,Z 384.523,A 0.000,B 0.000,C 90.000,E1 94.073} C_DIS
LIN {X 0.212,Y -478.339,Z 384.516,A 0.000,B 0.000,C 90.000,E1 92.808} C_DIS
LIN {X -0.019,Y -453.217,Z 384.497,A 0.000,B 0.000,C 90.000,E1 89.542} C_DIS
LIN {X -0.083,Y -433.993,Z 384.481,A 0.000,B 0.000,C 90.000,E1 86.674} C_DIS
LIN {X -0.115,Y -414.828,Z 384.464,A 0.000,B 0.000,C 90.000,E1 83.451} C_DIS
LIN {X -0.150,Y -402.673,Z 384.451,A 0.000,B 0.000,C 90.000,E1 81.254} C_DIS
LIN {X -0.027,Y -390.865,Z 384.439,A 0.000,B 0.000,C 90.000,E1 78.993} C_DIS
LIN {X -0.001,Y -380.553,Z 384.428,A 0.000,B 0.000,C 90.000,E1 76.992} C_DIS
LIN {X -0.088,Y -369.010,Z 384.415,A 0.000,B 0.000,C 90.000,E1 74.685} C_DIS
LIN {X -0.009,Y -357.617,Z 384.402,A 0.000,B 0.000,C 90.000,E1 72.308} C_DIS
LIN {X 0.108,Y -346.511,Z 384.388,A 0.000,B 0.000,C 90.000,E1 69.880} C_DIS
LIN {X 0.191,Y -334.318,Z 384.373,A 0.000,B 0.000,C 90.000,E1 67.102} C_DIS
LIN {X -0.144,Y -321.541,Z 384.356,A 0.000,B 0.000,C 90.000,E1 64.024} C_DIS
LIN {X 0.042,Y -308.457,Z 384.336,A 0.000,B 0.000,C 90.000,E1 60.461} C_DIS
LIN {X 0.140,Y -296.361,Z 384.316,A 0.000,B 0.000,C 90.000,E1 56.834} C_DIS
LIN {X 0.109,Y -286.294,Z 384.297,A 0.000,B 0.000,C 90.000,E1 53.497} C_DIS
LIN {X -0.018,Y -278.807,Z 384.282,A 0.000,B 0.000,C 90.000,E1 50.803} C_DIS
LIN {X 0.037,Y -273.235,Z 384.271,A 0.000,B 0.000,C 90.000,E1 48.728} C_DIS
LIN {X -0.058,Y -267.598,Z 384.259,A 0.000,B 0.000,C 90.000,E1 46.662} C_DIS
LIN {X 0.125,Y -261.846,Z 384.247,A 0.000,B 0.000,C 90.000,E1 44.514} C_DIS
LIN {X 0.018,Y -255.983,Z 384.236,A 0.000,B 0.000,C 90.000,E1 42.405} C_DIS
LIN {X -0.004,Y -249.971,Z 384.224,A 0.000,B 0.000,C 90.000,E1 40.253} C_DIS
LIN {X 0.083,Y -241.884,Z 384.207,A 0.000,B 0.000,C 90.000,E1 37.317} C_DIS
LIN {X -0.129,Y -234.197,Z 384.191,A 0.000,B 0.000,C 90.000,E1 34.405} C_DIS
LIN {X 0.056,Y -225.145,Z 384.170,A 0.000,B 0.000,C 90.000,E1 30.590} C_DIS
LIN {X 0.098,Y -218.422,Z 384.153,A 0.000,B 0.000,C 90.000,E1 27.513} C_DIS
LIN {X 0.014,Y -210.946,Z 384.131,A 0.000,B 0.000,C 90.000,E1 23.643} C_DIS
LIN {X 0.019,Y -205.733,Z 384.114,A 0.000,B 0.000,C 90.000,E1 20.482} C_DIS
LIN {X -0.021,Y -200.076,Z 384.092,A 0.000,B 0.000,C 90.000,E1 16.496} C_DIS
LIN {X 0.115,Y -195.357,Z 384.069,A 0.000,B 0.000,C 90.000,E1 12.411} C_DIS
LIN {X 0.058,Y -191.628,Z 384.046,A 0.000,B 0.000,C 90.000,E1 8.341} C_DIS
LIN {X -0.090,Y -188.872,Z 384.019,A 0.000,B 0.000,C 90.000,E1 3.440} C_DIS
LIN {X 0.021,Y -189.846,Z 383.942,A 0.000,B 0.000,C 90.000,E1 349.577} C_DIS
LIN {X 0.021,Y -192.917,Z 383.915,A 0.000,B 0.000,C 90.000,E1 344.629} C_DIS
LIN {X -0.034,Y -196.586,Z 383.892,A 0.000,B 0.000,C 90.000,E1 340.550} C_DIS
LIN {X -0.018,Y -201.405,Z 383.869,A 0.000,B 0.000,C 90.000,E1 336.485} C_DIS
LIN {X 0.032,Y -206.061,Z 383.851,A 0.000,B 0.000,C 90.000,E1 333.256} C_DIS
LIN {X 0.036,Y -212.725,Z 383.829,A 0.000,B 0.000,C 90.000,E1 329.282} C_DIS
LIN {X -0.048,Y -218.521,Z 383.812,A 0.000,B 0.000,C 90.000,E1 326.167} C_DIS
LIN {X 0.067,Y -226.305,Z 383.790,A 0.000,B 0.000,C 90.000,E1 322.271} C_DIS
LIN {X -0.002,Y -234.980,Z 383.769,A 0.000,B 0.000,C 90.000,E1 318.485} C_DIS
LIN {X 0.009,Y -244.025,Z 383.751,A 0.000,B 0.000,C 90.000,E1 315.121} C_DIS
LIN {X -0.054,Y -253.007,Z 383.734,A 0.000,B 0.000,C 90.000,E1 312.204} C_DIS
LIN {X 0.012,Y -264.328,Z 383.716,A 0.000,B 0.000,C 90.000,E1 308.955} C_DIS
LIN {X 0.028,Y -274.982,Z 383.701,A 0.000,B 0.000,C 90.000,E1 306.137} C_DIS
LIN {X 0.000,Y -289.012,Z 383.682,A 0.000,B 0.000,C 90.000,E1 302.704} C_DIS
LIN {X 0.094,Y -301.327,Z 383.667,A 0.000,B 0.000,C 90.000,E1 300.001} C_DIS
LIN {X -0.041,Y -316.741,Z 383.650,A 0.000,B 0.000,C 90.000,E1 297.078} C_DIS
LIN {X 0.057,Y -330.237,Z 383.638,A 0.000,B 0.000,C 90.000,E1 294.823} C_DIS
LIN {X 0.061,Y -349.574,Z 383.622,A 0.000,B 0.000,C 90.000,E1 292.025} C_DIS
LIN {X -0.012,Y -372.379,Z 383.606,A 0.000,B 0.000,C 90.000,E1 289.033} C_DIS
LIN {X 0.108,Y -389.885,Z 383.594,A 0.000,B 0.000,C 90.000,E1 286.985} C_DIS
LIN {X 0.123,Y -408.156,Z 383.584,A 0.000,B 0.000,C 90.000,E1 285.064} C_DIS
LIN {X 0.169,Y -423.822,Z 383.575,A 0.000,B 0.000,C 90.000,E1 283.480} C_DIS
LIN {X -0.064,Y -433.954,Z 383.569,A 0.000,B 0.000,C 90.000,E1 282.479} C_DIS
LIN {X 0.169,Y -441.229,Z 383.565,A 0.000,B 0.000,C 90.000,E1 281.658} C_DIS
LIN {X -0.045,Y -448.081,Z 383.560,A 0.000,B 0.000,C 90.000,E1 280.894} C_DIS
LIN {X -0.037,Y -456.400,Z 383.555,A 0.000,B 0.000,C 90.000,E1 279.849} C_DIS
LIN {X -0.139,Y -462.126,Z 383.550,A 0.000,B 0.000,C 90.000,E1 279.086} C_DIS
LIN {X -0.194,Y -470.760,Z 383.543,A 0.000,B 0.000,C 90.000,E1 277.814} C_DIS
LIN {X 0.017,Y -476.983,Z 383.538,A 0.000,B 0.000,C 90.000,E1 276.777} C_DIS
LIN {X -0.037,Y -481.147,Z 383.533,A 0.000,B 0.000,C 90.000,E1 276.030} C_DIS
LIN {X -0.003,Y -484.714,Z 383.529,A 0.000,B 0.000,C 90.000,E1 275.277} C_DIS
LIN {X 0.012,Y -487.483,Z 383.525,A 0.000,B 0.000,C 90.000,E1 274.531} C_DIS
LIN {X 0.207,Y -488.902,Z 383.522,A 0.000,B 0.000,C 90.000,E1 274.012} C_DIS
LIN {X -0.111,Y -489.957,Z 383.520,A 0.000,B 0.000,C 90.000,E1 273.555} C_DIS
LIN {X 0.100,Y -490.700,Z 383.517,A 0.000,B 0.000,C 90.000,E1 273.037} C_DIS
LIN {X -0.201,Y -491.131,Z 383.514,A 0.000,B 0.000,C 90.000,E1 272.579} C_DIS
LIN {X -0.004,Y -491.292,Z 383.511,A 0.000,B 0.000,C 90.000,E1 272.064} C_DIS
LIN {X 0.213,Y -491.085,Z 383.509,A 0.000,B 0.000,C 90.000,E1 271.547} C_DIS
LIN {X -0.077,Y -490.541,Z 383.506,A 0.000,B 0.000,C 90.000,E1 271.088} C_DIS
LIN {X 0.125,Y -489.573,Z 383.503,A 0.000,B 0.000,C 90.000,E1 270.573} C_DIS
LIN {X -0.165,Y -488.162,Z 383.501,A 0.000,B 0.000,C 90.000,E1 270.115} C_DIS
LIN {X -0.124,Y -484.889,Z 383.496,A 0.000,B 0.000,C 90.000,E1 269.370} C_DIS
LIN {X 0.210,Y -483.491,Z 383.495,A 0.000,B 0.000,C 90.000,E1 269.083} C_DIS
LIN {X -0.110,Y -479.970,Z 383.492,A 0.000,B 0.000,C 90.000,E1 268.625} C_DIS
LIN {X 0.048,Y -475.422,Z 383.490,A 0.000,B 0.000,C 90.000,E1 268.108} C_DIS
LIN {X -0.128,Y -472.669,Z 383.488,A 0.000,B 0.000,C 90.000,E1 267.879} C_DIS
LIN {X 0.166,Y -469.567,Z 383.487,A 0.000,B 0.000,C 90.000,E1 267.593} C_DIS
LIN {X -0.189,Y -466.529,Z 383.486,A 0.000,B 0.000,C 90.000,E1 267.421} C_DIS
LIN {X -0.113,Y -459.817,Z 383.483,A 0.000,B 0.000,C 90.000,E1 267.020} C_DIS
LIN {X 0.110,Y -452.834,Z 383.482,A 0.000,B 0.000,C 90.000,E1 266.674} C_DIS
LIN {X -0.123,Y -445.700,Z 383.480,A 0.000,B 0.000,C 90.000,E1 266.445} C_DIS
LIN {X 0.044,Y -438.146,Z 383.479,A 0.000,B 0.000,C 90.000,E1 266.216} C_DIS
LIN {X 0.142,Y -430.029,Z 383.478,A 0.000,B 0.000,C 90.000,E1 266.045} C_DIS
LIN {X 0.151,Y -420.831,Z 383.478,A 0.000,B 0.000,C 90.000,E1 265.931} C_DIS
LIN {X -0.148,Y -412.157,Z 383.477,A 0.000,B 0.000,C 90.000,E1 265.927} C_DIS
LIN {X 0.094,Y -180.916,Z 383.477,A 0.000,B 0.000,C 90.000,E1 265.869} C_DIS
LIN {X -0.043,Y -180.830,Z 383.472,A 0.000,B 0.000,C 90.000,E1 264.894} C_DIS
LIN {X 0.031,Y -178.867,Z 383.442,A 0.000,B 0.000,C 90.000,E1 259.634} C_DIS
LIN {X -0.068,Y -175.909,Z 383.414,A 0.000,B 0.000,C 90.000,E1 254.574} C_DIS
LIN {X -0.011,Y -174.597,Z 383.405,A 0.000,B 0.000,C 90.000,E1 252.851} C_DIS
LIN {X -0.085,Y -171.579,Z 383.381,A 0.000,B 0.000,C 90.000,E1 248.592} C_DIS
LIN {X -0.095,Y -167.802,Z 383.357,A 0.000,B 0.000,C 90.000,E1 244.280} C_DIS
LIN {X 0.070,Y -166.520,Z 383.347,A 0.000,B 0.000,C 90.000,E1 242.487} C_DIS
LIN {X 0.059,Y -162.521,Z 383.323,A 0.000,B 0.000,C 90.000,E1 238.122} C_DIS
LIN {X 0.030,Y -161.194,Z 383.313,A 0.000,B 0.000,C 90.000,E1 236.373} C_DIS
LIN {X -0.068,Y -157.204,Z 383.289,A 0.000,B 0.000,C 90.000,E1 231.984} C_DIS
LIN {X -0.045,Y -155.933,Z 383.279,A 0.000,B 0.000,C 90.000,E1 230.194} C_DIS
LIN {X -0.085,Y -152.184,Z 383.254,A 0.000,B 0.000,C 90.000,E1 225.729} C_DIS
LIN {X -0.064,Y -150.431,Z 383.239,A 0.000,B 0.000,C 90.000,E1 223.014} C_DIS
LIN {X -0.036,Y -147.159,Z 383.214,A 0.000,B 0.000,C 90.000,E1 218.463} C_DIS
LIN {X -0.068,Y -145.173,Z 383.193,A 0.000,B 0.000,C 90.000,E1 214.818} C_DIS
LIN {X -0.032,Y -142.323,Z 383.163,A 0.000,B 0.000,C 90.000,E1 209.283} C_DIS
LIN {X -0.038,Y -141.712,Z 383.152,A 0.000,B 0.000,C 90.000,E1 207.436} C_DIS
LIN {X 0.010,Y -139.472,Z 383.116,A 0.000,B 0.000,C 90.000,E1 200.918} C_DIS
LIN {X -0.068,Y -139.204,Z 383.106,A 0.000,B 0.000,C 90.000,E1 199.087} C_DIS
LIN {X -0.010,Y -138.330,Z 383.054,A 0.000,B 0.000,C 90.000,E1 189.726} C_DIS
LIN {X -0.007,Y -139.439,Z 383.007,A 0.000,B 0.000,C 90.000,E1 181.318} C_DIS
LIN {X -0.067,Y -140.971,Z 382.976,A 0.000,B 0.000,C 90.000,E1 175.755} C_DIS
LIN {X 0.024,Y -142.727,Z 382.956,A 0.000,B 0.000,C 90.000,E1 172.008} C_DIS
LIN {X -0.019,Y -145.112,Z 382.930,A 0.000,B 0.000,C 90.000,E1 167.409} C_DIS
LIN {X -0.024,Y -147.735,Z 382.910,A 0.000,B 0.000,C 90.000,E1 163.740} C_DIS
LIN {X 0.058,Y -150.399,Z 382.889,A 0.000,B 0.000,C 90.000,E1 160.061} C_DIS
LIN {X -0.067,Y -153.834,Z 382.869,A 0.000,B 0.000,C 90.000,E1 156.485} C_DIS
LIN {X -0.008,Y -157.245,Z 382.849,A 0.000,B 0.000,C 90.000,E1 152.871} C_DIS
LIN {X -0.068,Y -161.417,Z 382.829,A 0.000,B 0.000,C 90.000,E1 149.331} C_DIS
LIN {X -0.059,Y -165.619,Z 382.810,A 0.000,B 0.000,C 90.000,E1 145.801} C_DIS
LIN {X 0.061,Y -170.547,Z 382.790,A 0.000,B 0.000,C 90.000,E1 142.271} C_DIS
LIN {X -0.031,Y -175.426,Z 382.771,A 0.000,B 0.000,C 90.000,E1 138.852} C_DIS
LIN {X 0.086,Y -181.049,Z 382.752,A 0.000,B 0.000,C 90.000,E1 135.405} C_DIS
LIN {X -0.047,Y -186.484,Z 382.734,A 0.000,B 0.000,C 90.000,E1 132.081} C_DIS
LIN {X 0.020,Y -191.105,Z 382.720,A 0.000,B 0.000,C 90.000,E1 129.564} C_DIS
LIN {X -0.059,Y -196.899,Z 382.702,A 0.000,B 0.000,C 90.000,E1 126.297} C_DIS
LIN {X -0.024,Y -198.498,Z 382.697,A 0.000,B 0.000,C 90.000,E1 125.471} C_DIS
LIN {X 0.100,Y -298.212,Z 382.697,A 0.000,B 0.000,C 90.000,E1 125.438} C_DIS
LIN {X 0.021,Y -300.873,Z 382.697,A 0.000,B 0.000,C 90.000,E1 125.391} C_DIS
LIN {X -0.010,Y -306.537,Z 382.695,A 0.000,B 0.000,C 90.000,E1 125.025} C_DIS
LIN {X -0.043,Y -309.621,Z 382.693,A 0.000,B 0.000,C 90.000,E1 124.659} C_DIS
LIN {X 0.008,Y -311.567,Z 382.691,A 0.000,B 0.000,C 90.000,E1 124.326} C_DIS
LIN {X 0.062,Y -313.086,Z 382.689,A 0.000,B 0.000,C 90.000,E1 123.992} C_DIS
LIN {X -0.165,Y -318.636,Z 382.680,A 0.000,B 0.000,C 90.000,E1 122.418} C_DIS
LIN {X -0.095,Y -329.363,Z 382.664,A 0.000,B 0.000,C 90.000,E1 119.539} C_DIS
LIN {X 0.101,Y -341.473,Z 382.648,A 0.000,B 0.000,C 90.000,E1 116.693} C_DIS
LIN {X 0.004,Y -353.490,Z 382.635,A 0.000,B 0.000,C 90.000,E1 114.259} C_DIS
LIN {X 0.095,Y -366.776,Z 382.621,A 0.000,B 0.000,C 90.000,E1 111.844} C_DIS
LIN {X 0.043,Y -381.426,Z 382.608,A 0.000,B 0.000,C 90.000,E1 109.504} C_DIS
LIN {X -0.030,Y -397.551,Z 382.596,A 0.000,B 0.000,C 90.000,E1 107.221} C_DIS
LIN {X 0.197,Y -415.268,Z 382.583,A 0.000,B 0.000,C 90.000,E1 104.954} C_DIS
LIN {X -0.116,Y -434.644,Z 382.571,A 0.000,B 0.000,C 90.000,E1 102.827} C_DIS
LIN {X 0.113,Y -454.908,Z 382.560,A 0.000,B 0.000,C 90.000,E1 100.782} C_DIS
LIN {X -0.208,Y -475.706,Z 382.550,A 0.000,B 0.000,C 90.000,E1 98.973} C_DIS
LIN {X -0.014,Y -488.958,Z 382.544,A 0.000,B 0.000,C 90.000,E1 97.871} C_DIS
LIN {X 0.130,Y -491.218,Z 382.543,A 0.000,B 0.000,C 90.000,E1 97.644} C_DIS
LIN {X -0.147,Y -492.938,Z 382.541,A 0.000,B 0.000,C 90.000,E1 97.466} C_DIS
LIN {X 0.181,Y -494.478,Z 382.540,A 0.000,B 0.000,C 90.000,E1 97.182} C_DIS
LIN {X 0.082,Y -495.629,Z 382.539,A 0.000,B 0.000,C 90.000,E1 96.947} C_DIS
LIN {X -0.161,Y -497.001,Z 382.536,A 0.000,B 0.000,C 90.000,E1 96.486} C_DIS
LIN {X 0.096,Y -497.329,Z 382.533,A 0.000,B 0.000,C 90.000,E1 95.967} C_DIS
LIN {X -0.182,Y -496.661,Z 382.530,A 0.000,B 0.000,C 90.000,E1 95.511} C_DIS
LIN {X 0.085,Y -494.887,Z 382.528,A 0.000,B 0.000,C 90.000,E1 94.992} C_DIS
LIN {X -0.009,Y -493.478,Z 382.526,A 0.000,B 0.000,C 90.000,E1 94.759} C_DIS
LIN {X 0.094,Y -488.098,Z 382.522,A 0.000,B 0.000,C 90.000,E1 94.012} C_DIS
LIN {X -0.183,Y -478.287,Z 382.515,A 0.000,B 0.000,C 90.000,E1 92.808} C_DIS
LIN {X 0.063,Y -453.161,Z 382.497,A 0.000,B 0.000,C 90.000,E1 89.484} C_DIS
LIN {X -0.195,Y -435.597,Z 382.483,A 0.000,B 0.000,C 90.000,E1 86.906} C_DIS
LIN {X -0.183,Y -416.308,Z 382.465,A 0.000,B 0.000,C 90.000,E1 83.685} C_DIS
LIN {X -0.189,Y -404.160,Z 382.453,A 0.000,B 0.000,C 90.000,E1 81.489} C_DIS
LIN {X 0.039,Y -392.319,Z 382.440,A 0.000,B 0.000,C 90.000,E1 79.218} C_DIS
LIN {X 0.020,Y -382.025,Z 382.429,A 0.000,B 0.000,C 90.000,E1 77.229} C_DIS
LIN {X -0.131,Y -370.447,Z 382.416,A 0.000,B 0.000,C 90.000,E1 74.936} C_DIS
LIN {X 0.081,Y -359.017,Z 382.403,A 0.000,B 0.000,C 90.000,E1 72.543} C_DIS
LIN {X 0.116,Y -347.840,Z 382.390,A 0.000,B 0.000,C 90.000,E1 70.134} C_DIS
LIN {X -0.083,Y -336.915,Z 382.376,A 0.000,B 0.000,C 90.000,E1 67.720} C_DIS
LIN {X -0.032,Y -323.963,Z 382.359,A 0.000,B 0.000,C 90.000,E1 64.588} C_DIS
LIN {X 0.092,Y -310.697,Z 382.339,A 0.000,B 0.000,C 90.000,E1 61.051} C_DIS
LIN {X 0.073,Y -299.473,Z 382.321,A 0.000,B 0.000,C 90.000,E1 57.788} C_DIS
LIN {X -0.024,Y -289.170,Z 382.303,A 0.000,B 0.000,C 90.000,E1 54.482} C_DIS
LIN {X 0.006,Y -279.675,Z 382.284,A 0.000,B 0.000,C 90.000,E1 51.090} C_DIS
LIN {X 0.079,Y -274.145,Z 382.272,A 0.000,B 0.000,C 90.000,E1 49.013} C_DIS
LIN {X 0.016,Y -268.510,Z 382.261,A 0.000,B 0.000,C 90.000,E1 46.944} C_DIS
LIN {X 0.022,Y -262.763,Z 382.249,A 0.000,B 0.000,C 90.000,E1 44.838} C_DIS
LIN {X 0.110,Y -256.969,Z 382.237,A 0.000,B 0.000,C 90.000,E1 42.690} C_DIS
LIN {X 0.100,Y -250.971,Z 382.225,A 0.000,B 0.000,C 90.000,E1 40.539} C_DIS
LIN {X 0.013,Y -242.875,Z 382.209,A 0.000,B 0.000,C 90.000,E1 37.649} C_DIS
LIN {X 0.015,Y -235.154,Z 382.193,A 0.000,B 0.000,C 90.000,E1 34.692} C_DIS
LIN {X 0.035,Y -226.025,Z 382.172,A 0.000,B 0.000,C 90.000,E1 30.924} C_DIS
LIN {X -0.093,Y -219.213,Z 382.155,A 0.000,B 0.000,C 90.000,E1 27.897} C_DIS
LIN {X -0.061,Y -211.619,Z 382.133,A 0.000,B 0.000,C 90.000,E1 24.003} C_DIS
LIN {X -0.041,Y -206.297,Z 382.116,A 0.000,B 0.000,C 90.000,E1 20.844} C_DIS
LIN {X -0.064,Y -200.531,Z 382.094,A 0.000,B 0.000,C 90.000,E1 16.858} C_DIS
LIN {X -0.098,Y -195.705,Z 382.071,A 0.000,B 0.000,C 90.000,E1 12.827} C_DIS
LIN {X -0.104,Y -191.857,Z 382.048,A 0.000,B 0.000,C 90.000,E1 8.746} C_DIS
LIN {X -0.037,Y -188.984,Z 382.021,A 0.000,B 0.000,C 90.000,E1 3.784} C_DIS
LIN {X -0.006,Y -190.154,Z 381.938,A 0.000,B 0.000,C 90.000,E1 348.757} C_DIS
LIN {X 0.057,Y -193.467,Z 381.910,A 0.000,B 0.000,C 90.000,E1 343.795} C_DIS
LIN {X 0.079,Y -197.360,Z 381.887,A 0.000,B 0.000,C 90.000,E1 339.699} C_DIS
LIN {X 0.014,Y -202.411,Z 381.865,A 0.000,B 0.000,C 90.000,E1 335.665} C_DIS
LIN {X -0.097,Y -207.245,Z 381.847,A 0.000,B 0.000,C 90.000,E1 332.487} C_DIS
LIN {X 0.042,Y -214.058,Z 381.825,A 0.000,B 0.000,C 90.000,E1 328.486} C_DIS
LIN {X -0.060,Y -221.420,Z 381.803,A 0.000,B 0.000,C 90.000,E1 324.609} C_DIS
LIN {X -0.091,Y -227.905,Z 381.786,A 0.000,B 0.000,C 90.000,E1 321.537} C_DIS
LIN {X -0.036,Y -234.903,Z 381.769,A 0.000,B 0.000,C 90.000,E1 318.485} C_DIS
LIN {X -0.027,Y -243.946,Z 381.751,A 0.000,B 0.000,C 90.000,E1 315.121} C_DIS
LIN {X 0.080,Y -251.755,Z 381.736,A 0.000,B 0.000,C 90.000,E1 312.528} C_DIS
LIN {X 0.125,Y -262.992,Z 381.718,A 0.000,B 0.000,C 90.000,E1 309.277} C_DIS
LIN {X -0.100,Y -273.580,Z 381.703,A 0.000,B 0.000,C 90.000,E1 306.503} C_DIS
LIN {X -0.019,Y -287.449,Z 381.684,A 0.000,B 0.000,C 90.000,E1 303.038} C_DIS
LIN {X 0.038,Y -301.296,Z 381.667,A 0.000,B 0.000,C 90.000,E1 300.001} C_DIS
LIN {X -0.011,Y -314.974,Z 381.652,A 0.000,B 0.000,C 90.000,E1 297.385} C_DIS
LIN {X -0.040,Y -326.334,Z 381.641,A 0.000,B 0.000,C 90.000,E1 295.463} C_DIS
LIN {X -0.106,Y -336.673,Z 381.633,A 0.000,B 0.000,C 90.000,E1 293.898} C_DIS
LIN {X 0.050,Y -354.229,Z 381.619,A 0.000,B 0.000,C 90.000,E1 291.408} C_DIS
LIN {X -0.069,Y -372.597,Z 381.606,A 0.000,B 0.000,C 90.000,E1 289.033} C_DIS
LIN {X -0.129,Y -389.912,Z 381.595,A 0.000,B 0.000,C 90.000,E1 287.040} C_DIS
LIN {X -0.109,Y -407.988,Z 381.584,A 0.000,B 0.000,C 90.000,E1 285.134} C_DIS
LIN {X 0.075,Y -423.549,Z 381.575,A 0.000,B 0.000,C 90.000,E1 283.536} C_DIS
LIN {X -0.198,Y -433.719,Z 381.569,A 0.000,B 0.000,C 90.000,E1 282.535} C_DIS
LIN {X 0.013,Y -441.010,Z 381.565,A 0.000,B 0.000,C 90.000,E1 281.715} C_DIS
LIN {X 0.021,Y -449.982,Z 381.559,A 0.000,B 0.000,C 90.000,E1 280.658} C_DIS
LIN {X 0.052,Y -458.125,Z 381.553,A 0.000,B 0.000,C 90.000,E1 279.613} C_DIS
LIN {X -0.104,Y -463.678,Z 381.549,A 0.000,B 0.000,C 90.000,E1 278.859} C_DIS
LIN {X 0.089,Y -470.501,Z 381.543,A 0.000,B 0.000,C 90.000,E1 277.814} C_DIS
LIN {X -0.172,Y -476.745,Z 381.538,A 0.000,B 0.000,C 90.000,E1 276.834} C_DIS
LIN {X 0.113,Y -482.222,Z 381.532,A 0.000,B 0.000,C 90.000,E1 275.796} C_DIS
LIN {X 0.107,Y -485.531,Z 381.528,A 0.000,B 0.000,C 90.000,E1 275.049} C_DIS
LIN {X -0.190,Y -487.312,Z 381.525,A 0.000,B 0.000,C 90.000,E1 274.588} C_DIS
LIN {X -0.032,Y -488.757,Z 381.523,A 0.000,B 0.000,C 90.000,E1 274.073} C_DIS
LIN {X 0.173,Y -489.826,Z 381.520,A 0.000,B 0.000,C 90.000,E1 273.555} C_DIS
LIN {X -0.108,Y -490.606,Z 381.517,A 0.000,B 0.000,C 90.000,E1 273.094} C_DIS
LIN {X 0.082,Y -491.059,Z 381.514,A 0.000,B 0.000,C 90.000,E1 272.579} C_DIS
LIN {X -0.212,Y -491.244,Z 381.512,A 0.000,B 0.000,C 90.000,E1 272.121} C_DIS
LIN {X 0.003,Y -491.076,Z 381.509,A 0.000,B 0.000,C 90.000,E1 271.604} C_DIS
LIN {X 0.204,Y -490.550,Z 381.506,A 0.000,B 0.000,C 90.000,E1 271.088} C_DIS
LIN {X -0.084,Y -489.598,Z 381.503,A 0.000,B 0.000,C 90.000,E1 270.630} C_DIS
LIN {X 0.114,Y -488.202,Z 381.501,A 0.000,B 0.000,C 90.000,E1 270.115} C_DIS
LIN {X -0.180,Y -486.275,Z 381.498,A 0.000,B 0.000,C 90.000,E1 269.656} C_DIS
LIN {X 0.155,Y -485.088,Z 381.497,A 0.000,B 0.000,C 90.000,E1 269.370} C_DIS
LIN {X -0.155,Y -482.116,Z 381.494,A 0.000,B 0.000,C 90.000,E1 268.912} C_DIS
LIN {X -0.001,Y -478.196,Z 381.491,A 0.000,B 0.000,C 90.000,E1 268.396} C_DIS
LIN {X 0.146,Y -473.156,Z 381.488,A 0.000,B 0.000,C 90.000,E1 267.879} C_DIS
LIN {X -0.029,Y -470.132,Z 381.487,A 0.000,B 0.000,C 90.000,E1 267.650} C_DIS
LIN {X 0.054,Y -467.103,Z 381.486,A 0.000,B 0.000,C 90.000,E1 267.421} C_DIS
LIN {X 0.077,Y -460.452,Z 381.483,A 0.000,B 0.000,C 90.000,E1 267.020} C_DIS
LIN {X -0.210,Y -453.462,Z 381.482,A 0.000,B 0.000,C 90.000,E1 266.731} C_DIS
LIN {X -0.052,Y -446.261,Z 381.480,A 0.000,B 0.000,C 90.000,E1 266.445} C_DIS
LIN {X 0.061,Y -438.588,Z 381.479,A 0.000,B 0.000,C 90.000,E1 266.216} C_DIS
LIN {X 0.125,Y -430.245,Z 381.478,A 0.000,B 0.000,C 90.000,E1 266.045} C_DIS
LIN {X 0.126,Y -420.934,Z 381.477,A 0.000,B 0.000,C 90.000,E1 265.931} C_DIS
LIN {X -0.179,Y -411.735,Z 381.477,A 0.000,B 0.000,C 90.000,E1 265.927} C_DIS
LIN {X 0.081,Y -180.916,Z 381.477,A 0.000,B 0.000,C 90.000,E1 265.869} C_DIS
LIN {X -0.057,Y -180.829,Z 381.472,A 0.000,B 0.000,C 90.000,E1 264.894} C_DIS
LIN {X 0.017,Y -178.864,Z 381.442,A 0.000,B 0.000,C 90.000,E1 259.634} C_DIS
LIN {X -0.082,Y -175.908,Z 381.414,A 0.000,B 0.000,C 90.000,E1 254.574} C_DIS
LIN {X 0.026,Y -174.593,Z 381.405,A 0.000,B 0.000,C 90.000,E1 252.834} C_DIS
LIN {X 0.061,Y -171.575,Z 381.381,A 0.000,B 0.000,C 90.000,E1 248.539} C_DIS
LIN {X 0.043,Y -167.798,Z 381.357,A 0.000,B 0.000,C 90.000,E1 244.229} C_DIS
LIN {X 0.057,Y -166.515,Z 381.347,A 0.000,B 0.000,C 90.000,E1 242.487} C_DIS
LIN {X 0.052,Y -163.223,Z 381.328,A 0.000,B 0.000,C 90.000,E1 238.997} C_DIS
LIN {X 0.017,Y -161.189,Z 381.313,A 0.000,B 0.000,C 90.000,E1 236.373} C_DIS
LIN {X -0.081,Y -157.201,Z 381.289,A 0.000,B 0.000,C 90.000,E1 231.984} C_DIS
LIN {X -0.058,Y -155.929,Z 381.279,A 0.000,B 0.000,C 90.000,E1 230.194} C_DIS
LIN {X 0.012,Y -152.181,Z 381.254,A 0.000,B 0.000,C 90.000,E1 225.688} C_DIS
LIN {X 0.027,Y -150.428,Z 381.239,A 0.000,B 0.000,C 90.000,E1 222.975} C_DIS
LIN {X -0.048,Y -147.155,Z 381.214,A 0.000,B 0.000,C 90.000,E1 218.463} C_DIS
LIN {X -0.080,Y -145.171,Z 381.193,A 0.000,B 0.000,C 90.000,E1 214.818} C_DIS
LIN {X -0.045,Y -142.320,Z 381.163,A 0.000,B 0.000,C 90.000,E1 209.283} C_DIS
LIN {X 0.075,Y -141.710,Z 381.152,A 0.000,B 0.000,C 90.000,E1 207.385} C_DIS
LIN {X -0.002,Y -139.471,Z 381.116,A 0.000,B 0.000,C 90.000,E1 200.918} C_DIS
LIN {X 0.052,Y -139.203,Z 381.106,A 0.000,B 0.000,C 90.000,E1 199.033} C_DIS
LIN {X -0.022,Y -138.328,Z 381.054,A 0.000,B 0.000,C 90.000,E1 189.726} C_DIS
LIN {X -0.019,Y -139.439,Z 381.007,A 0.000,B 0.000,C 90.000,E1 181.318} C_DIS
LIN {X 0.061,Y -140.973,Z 380.976,A 0.000,B 0.000,C 90.000,E1 175.698} C_DIS
LIN {X 0.011,Y -142.729,Z 380.956,A 0.000,B 0.000,C 90.000,E1 172.008} C_DIS
LIN {X -0.031,Y -145.115,Z 380.930,A 0.000,B 0.000,C 90.000,E1 167.409} C_DIS
LIN {X -0.037,Y -147.739,Z 380.910,A 0.000,B 0.000,C 90.000,E1 163.740} C_DIS
LIN {X 0.045,Y -150.403,Z 380.889,A 0.000,B 0.000,C 90.000,E1 160.061} C_DIS
LIN {X -0.081,Y -153.839,Z 380.869,A 0.000,B 0.000,C 90.000,E1 156.485} C_DIS
LIN {X -0.022,Y -157.250,Z 380.849,A 0.000,B 0.000,C 90.000,E1 152.871} C_DIS
LIN {X 0.057,Y -161.423,Z 380.829,A 0.000,B 0.000,C 90.000,E1 149.282} C_DIS
LIN {X -0.073,Y -165.625,Z 380.810,A 0.000,B 0.000,C 90.000,E1 145.801} C_DIS
LIN {X 0.047,Y -170.554,Z 380.790,A 0.000,B 0.000,C 90.000,E1 142.271} C_DIS
LIN {X -0.045,Y -175.433,Z 380.771,A 0.000,B 0.000,C 90.000,E1 138.852} C_DIS
LIN {X 0.072,Y -181.055,Z 380.752,A 0.000,B 0.000,C 90.000,E1 135.405} C_DIS
LIN {X -0.062,Y -186.492,Z 380.734,A 0.000,B 0.000,C 90.000,E1 132.081} C_DIS
LIN {X 0.005,Y -191.113,Z 380.720,A 0.000,B 0.000,C 90.000,E1 129.564} C_DIS
LIN {X -0.074,Y -196.907,Z 380.702,A 0.000,B 0.000,C 90.000,E1 126.297} C_DIS
LIN {X -0.055,Y -198.582,Z 380.697,A 0.000,B 0.000,C 90.000,E1 125.438} C_DIS
LIN {X 0.106,Y -297.659,Z 380.697,A 0.000,B 0.000,C 90.000,E1 125.391} C_DIS
LIN {X -0.003,Y -299.371,Z 380.697,A 0.000,B 0.000,C 90.000,E1 125.391} C_DIS
LIN {X 0.107,Y -303.804,Z 380.696,A 0.000,B 0.000,C 90.000,E1 125.185} C_DIS
LIN {X -0.033,Y -306.193,Z 380.695,A 0.000,B 0.000,C 90.000,E1 125.025} C_DIS
LIN {X -0.067,Y -309.441,Z 380.692,A 0.000,B 0.000,C 90.000,E1 124.659} C_DIS
LIN {X 0.048,Y -311.398,Z 380.691,A 0.000,B 0.000,C 90.000,E1 124.326} C_DIS
LIN {X -0.093,Y -312.934,Z 380.689,A 0.000,B 0.000,C 90.000,E1 124.040} C_DIS
LIN {X 0.010,Y -315.269,Z 380.685,A 0.000,B 0.000,C 90.000,E1 123.372} C_DIS
LIN {X 0.158,Y -325.545,Z 380.669,A 0.000,B 0.000,C 90.000,E1 120.463} C_DIS
LIN {X 0.105,Y -337.175,Z 380.654,A 0.000,B 0.000,C 90.000,E1 117.641} C_DIS
LIN {X -0.085,Y -350.259,Z 380.638,A 0.000,B 0.000,C 90.000,E1 114.899} C_DIS
LIN {X 0.064,Y -363.210,Z 380.625,A 0.000,B 0.000,C 90.000,E1 112.461} C_DIS
LIN {X -0.076,Y -377.500,Z 380.612,A 0.000,B 0.000,C 90.000,E1 110.120} C_DIS
LIN {X -0.125,Y -393.234,Z 380.599,A 0.000,B 0.000,C 90.000,E1 107.819} C_DIS
LIN {X -0.014,Y -410.528,Z 380.586,A 0.000,B 0.000,C 90.000,E1 105.552} C_DIS
LIN {X 0.028,Y -429.504,Z 380.574,A 0.000,B 0.000,C 90.000,E1 103.355} C_DIS
LIN {X -0.014,Y -449.620,Z 380.563,A 0.000,B 0.000,C 90.000,E1 101.299} C_DIS
LIN {X 0.243,Y -470.287,Z 380.552,A 0.000,B 0.000,C 90.000,E1 99.378} C_DIS
LIN {X 0.082,Y -488.783,Z 380.544,A 0.000,B 0.000,C 90.000,E1 97.871} C_DIS
LIN {X -0.238,Y -491.114,Z 380.543,A 0.000,B 0.000,C 90.000,E1 97.701} C_DIS
LIN {X -0.007,Y -492.884,Z 380.541,A 0.000,B 0.000,C 90.000,E1 97.466} C_DIS
LIN {X -0.169,Y -494.486,Z 380.540,A 0.000,B 0.000,C 90.000,E1 97.239} C_DIS
LIN {X 0.222,Y -495.686,Z 380.539,A 0.000,B 0.000,C 90.000,E1 96.947} C_DIS
LIN {X -0.020,Y -497.136,Z 380.536,A 0.000,B 0.000,C 90.000,E1 96.486} C_DIS
LIN {X 0.237,Y -497.530,Z 380.533,A 0.000,B 0.000,C 90.000,E1 95.967} C_DIS
LIN {X -0.041,Y -496.931,Z 380.531,A 0.000,B 0.000,C 90.000,E1 95.511} C_DIS
LIN {X 0.228,Y -495.238,Z 380.528,A 0.000,B 0.000,C 90.000,E1 94.992} C_DIS
LIN {X 0.134,Y -493.884,Z 380.527,A 0.000,B 0.000,C 90.000,E1 94.759} C_DIS
LIN {X 0.239,Y -488.548,Z 380.522,A 0.000,B 0.000,C 90.000,E1 94.012} C_DIS
LIN {X 0.133,Y -480.768,Z 380.517,A 0.000,B 0.000,C 90.000,E1 93.037} C_DIS
LIN {X 0.208,Y -457.289,Z 380.500,A 0.000,B 0.000,C 90.000,E1 90.000} C_DIS
LIN {X -0.032,Y -435.971,Z 380.483,A 0.000,B 0.000,C 90.000,E1 86.906} C_DIS
LIN {X 0.117,Y -415.124,Z 380.463,A 0.000,B 0.000,C 90.000,E1 83.394} C_DIS
LIN {X 0.081,Y -403.024,Z 380.451,A 0.000,B 0.000,C 90.000,E1 81.197} C_DIS
LIN {X -0.182,Y -391.209,Z 380.439,A 0.000,B 0.000,C 90.000,E1 78.993} C_DIS
LIN {X -0.140,Y -380.942,Z 380.428,A 0.000,B 0.000,C 90.000,E1 76.992} C_DIS
LIN {X 0.143,Y -369.390,Z 380.415,A 0.000,B 0.000,C 90.000,E1 74.629} C_DIS
LIN {X -0.121,Y -357.958,Z 380.402,A 0.000,B 0.000,C 90.000,E1 72.308} C_DIS
LIN {X 0.007,Y -346.764,Z 380.388,A 0.000,B 0.000,C 90.000,E1 69.880} C_DIS
LIN {X 0.095,Y -334.528,Z 380.373,A 0.000,B 0.000,C 90.000,E1 67.102} C_DIS
LIN {X 0.059,Y -321.695,Z 380.355,A 0.000,B 0.000,C 90.000,E1 63.973} C_DIS
LIN {X -0.032,Y -308.613,Z 380.336,A 0.000,B 0.000,C 90.000,E1 60.461} C_DIS
LIN {X 0.053,Y -297.571,Z 380.318,A 0.000,B 0.000,C 90.000,E1 57.168} C_DIS
LIN {X 0.067,Y -287.427,Z 380.299,A 0.000,B 0.000,C 90.000,E1 53.829} C_DIS
LIN {X 0.043,Y -278.067,Z 380.280,A 0.000,B 0.000,C 90.000,E1 50.436} C_DIS
LIN {X -0.125,Y -272.486,Z 380.269,A 0.000,B 0.000,C 90.000,E1 48.405} C_DIS
LIN {X -0.033,Y -266.812,Z 380.257,A 0.000,B 0.000,C 90.000,E1 46.296} C_DIS
LIN {X -0.054,Y -261.051,Z 380.245,A 0.000,B 0.000,C 90.000,E1 44.190} C_DIS
LIN {X -0.002,Y -255.229,Z 380.234,A 0.000,B 0.000,C 90.000,E1 42.043} C_DIS
LIN {X -0.016,Y -249.197,Z 380.222,A 0.000,B 0.000,C 90.000,E1 39.886} C_DIS
LIN {X 0.034,Y -239.234,Z 380.201,A 0.000,B 0.000,C 90.000,E1 36.217} C_DIS
LIN {X 0.005,Y -231.683,Z 380.185,A 0.000,B 0.000,C 90.000,E1 33.245} C_DIS
LIN {X -0.011,Y -222.795,Z 380.164,A 0.000,B 0.000,C 90.000,E1 29.461} C_DIS
LIN {X 0.064,Y -216.254,Z 380.147,A 0.000,B 0.000,C 90.000,E1 26.360} C_DIS
LIN {X -0.019,Y -210.346,Z 380.129,A 0.000,B 0.000,C 90.000,E1 23.259} C_DIS
LIN {X -0.105,Y -205.182,Z 380.112,A 0.000,B 0.000,C 90.000,E1 20.120} C_DIS
LIN {X 0.034,Y -199.552,Z 380.089,A 0.000,B 0.000,C 90.000,E1 16.079} C_DIS
LIN {X -0.081,Y -194.899,Z 380.067,A 0.000,B 0.000,C 90.000,E1 12.063} C_DIS
LIN {X 0.042,Y -191.255,Z 380.044,A 0.000,B 0.000,C 90.000,E1 7.936} C_DIS
LIN {X -0.019,Y -188.405,Z 380.012,A 0.000,B 0.000,C 90.000,E1 2.178} C_DIS
LIN {X 0.013,Y -189.658,Z 379.942,A 0.000,B 0.000,C 90.000,E1 349.577} C_DIS
LIN {X 0.005,Y -192.729,Z 379.915,A 0.000,B 0.000,C 90.000,E1 344.629} C_DIS
LIN {X -0.057,Y -196.403,Z 379.892,A 0.000,B 0.000,C 90.000,E1 340.550} C_DIS
LIN {X -0.046,Y -201.218,Z 379.869,A 0.000,B 0.000,C 90.000,E1 336.485} C_DIS
LIN {X -0.002,Y -205.842,Z 379.851,A 0.000,B 0.000,C 90.000,E1 333.256} C_DIS
LIN {X -0.006,Y -212.545,Z 379.829,A 0.000,B 0.000,C 90.000,E1 329.282} C_DIS
LIN {X -0.096,Y -219.796,Z 379.808,A 0.000,B 0.000,C 90.000,E1 325.388} C_DIS
LIN {X 0.010,Y -226.113,Z 379.790,A 0.000,B 0.000,C 90.000,E1 322.271} C_DIS
LIN {X -0.067,Y -234.822,Z 379.769,A 0.000,B 0.000,C 90.000,E1 318.485} C_DIS
LIN {X 0.110,Y -243.875,Z 379.751,A 0.000,B 0.000,C 90.000,E1 315.081} C_DIS
LIN {X 0.042,Y -251.687,Z 379.736,A 0.000,B 0.000,C 90.000,E1 312.528} C_DIS
LIN {X 0.083,Y -262.942,Z 379.718,A 0.000,B 0.000,C 90.000,E1 309.277} C_DIS
LIN {X 0.076,Y -273.524,Z 379.703,A 0.000,B 0.000,C 90.000,E1 306.457} C_DIS
LIN {X -0.036,Y -285.900,Z 379.685,A 0.000,B 0.000,C 90.000,E1 303.372} C_DIS
LIN {X -0.020,Y -299.651,Z 379.669,A 0.000,B 0.000,C 90.000,E1 300.335} C_DIS
LIN {X -0.066,Y -315.015,Z 379.652,A 0.000,B 0.000,C 90.000,E1 297.385} C_DIS
LIN {X -0.096,Y -326.436,Z 379.641,A 0.000,B 0.000,C 90.000,E1 295.463} C_DIS
LIN {X -0.162,Y -336.812,Z 379.633,A 0.000,B 0.000,C 90.000,E1 293.898} C_DIS
LIN {X -0.005,Y -354.421,Z 379.619,A 0.000,B 0.000,C 90.000,E1 291.408} C_DIS
LIN {X -0.032,Y -375.226,Z 379.604,A 0.000,B 0.000,C 90.000,E1 288.725} C_DIS
LIN {X -0.151,Y -397.935,Z 379.590,A 0.000,B 0.000,C 90.000,E1 286.205} C_DIS
LIN {X -0.132,Y -415.832,Z 379.580,A 0.000,B 0.000,C 90.000,E1 284.356} C_DIS
LIN {X -0.124,Y -428.645,Z 379.572,A 0.000,B 0.000,C 90.000,E1 283.063} C_DIS
LIN {X 0.183,Y -436.087,Z 379.568,A 0.000,B 0.000,C 90.000,E1 282.243} C_DIS
LIN {X -0.064,Y -443.233,Z 379.564,A 0.000,B 0.000,C 90.000,E1 281.478} C_DIS
LIN {X 0.168,Y -449.866,Z 379.559,A 0.000,B 0.000,C 90.000,E1 280.658} C_DIS
LIN {X 0.200,Y -458.005,Z 379.554,A 0.000,B 0.000,C 90.000,E1 279.613} C_DIS
LIN {X -0.129,Y -465.289,Z 379.548,A 0.000,B 0.000,C 90.000,E1 278.624} C_DIS
LIN {X 0.016,Y -471.993,Z 379.542,A 0.000,B 0.000,C 90.000,E1 277.587} C_DIS
LIN {X -0.226,Y -478.058,Z 379.537,A 0.000,B 0.000,C 90.000,E1 276.606} C_DIS
LIN {X -0.217,Y -482.062,Z 379.532,A 0.000,B 0.000,C 90.000,E1 275.853} C_DIS
LIN {X -0.051,Y -484.397,Z 379.530,A 0.000,B 0.000,C 90.000,E1 275.334} C_DIS
LIN {X -0.040,Y -487.221,Z 379.525,A 0.000,B 0.000,C 90.000,E1 274.588} C_DIS
LIN {X 0.117,Y -488.649,Z 379.523,A 0.000,B 0.000,C 90.000,E1 274.073} C_DIS
LIN {X -0.167,Y -489.723,Z 379.520,A 0.000,B 0.000,C 90.000,E1 273.612} C_DIS
LIN {X 0.041,Y -490.504,Z 379.517,A 0.000,B 0.000,C 90.000,E1 273.094} C_DIS
LIN {X 0.230,Y -490.968,Z 379.514,A 0.000,B 0.000,C 90.000,E1 272.579} C_DIS
LIN {X -0.065,Y -491.161,Z 379.512,A 0.000,B 0.000,C 90.000,E1 272.121} C_DIS
LIN {X 0.151,Y -491.017,Z 379.509,A 0.000,B 0.000,C 90.000,E1 271.604} C_DIS
LIN {X -0.139,Y -490.519,Z 379.506,A 0.000,B 0.000,C 90.000,E1 271.146} C_DIS
LIN {X 0.062,Y -489.600,Z 379.504,A 0.000,B 0.000,C 90.000,E1 270.630} C_DIS
LIN {X -0.229,Y -488.258,Z 379.501,A 0.000,B 0.000,C 90.000,E1 270.172} C_DIS
LIN {X -0.036,Y -486.327,Z 379.498,A 0.000,B 0.000,C 90.000,E1 269.656} C_DIS
LIN {X -0.186,Y -485.176,Z 379.497,A 0.000,B 0.000,C 90.000,E1 269.427} C_DIS
LIN {X -0.012,Y -482.213,Z 379.494,A 0.000,B 0.000,C 90.000,E1 268.912} C_DIS
LIN {X -0.170,Y -480.440,Z 379.493,A 0.000,B 0.000,C 90.000,E1 268.682} C_DIS
LIN {X -0.009,Y -476.075,Z 379.490,A 0.000,B 0.000,C 90.000,E1 268.165} C_DIS
LIN {X -0.183,Y -473.414,Z 379.488,A 0.000,B 0.000,C 90.000,E1 267.936} C_DIS
LIN {X 0.114,Y -470.424,Z 379.487,A 0.000,B 0.000,C 90.000,E1 267.650} C_DIS
LIN {X 0.183,Y -467.458,Z 379.486,A 0.000,B 0.000,C 90.000,E1 267.421} C_DIS
LIN {X -0.214,Y -464.063,Z 379.485,A 0.000,B 0.000,C 90.000,E1 267.249} C_DIS
LIN {X 0.077,Y -457.140,Z 379.483,A 0.000,B 0.000,C 90.000,E1 266.846} C_DIS
LIN {X -0.005,Y -449.977,Z 379.481,A 0.000,B 0.000,C 90.000,E1 266.560} C_DIS
LIN {X -0.100,Y -442.539,Z 379.480,A 0.000,B 0.000,C 90.000,E1 266.331} C_DIS
LIN {X 0.206,Y -434.607,Z 379.478,A 0.000,B 0.000,C 90.000,E1 266.102} C_DIS
LIN {X 0.018,Y -425.804,Z 379.478,A 0.000,B 0.000,C 90.000,E1 265.988} C_DIS
LIN {X -0.051,Y -417.858,Z 379.477,A 0.000,B 0.000,C 90.000,E1 265.927} C_DIS
LIN {X -0.189,Y -411.938,Z 379.477,A 0.000,B 0.000,C 90.000,E1 265.927} C_DIS
LIN {X 0.077,Y -180.916,Z 379.477,A 0.000,B 0.000,C 90.000,E1 265.869} C_DIS
LIN {X -0.060,Y -180.829,Z 379.472,A 0.000,B 0.000,C 90.000,E1 264.894} C_DIS
LIN {X 0.014,Y -178.864,Z 379.442,A 0.000,B 0.000,C 90.000,E1 259.634} C_DIS
LIN {X -0.085,Y -175.907,Z 379.414,A 0.000,B 0.000,C 90.000,E1 254.574} C_DIS
LIN {X 0.023,Y -174.592,Z 379.405,A 0.000,B 0.000,C 90.000,E1 252.834} C_DIS
LIN {X 0.058,Y -171.575,Z 379.381,A 0.000,B 0.000,C 90.000,E1 248.539} C_DIS
LIN {X 0.039,Y -167.797,Z 379.357,A 0.000,B 0.000,C 90.000,E1 244.229} C_DIS
LIN {X 0.054,Y -166.515,Z 379.347,A 0.000,B 0.000,C 90.000,E1 242.487} C_DIS
LIN {X 0.049,Y -163.223,Z 379.328,A 0.000,B 0.000,C 90.000,E1 238.997} C_DIS
LIN {X 0.014,Y -161.189,Z 379.313,A 0.000,B 0.000,C 90.000,E1 236.373} C_DIS
LIN {X -0.084,Y -157.200,Z 379.289,A 0.000,B 0.000,C 90.000,E1 231.984} C_DIS
LIN {X -0.060,Y -155.928,Z 379.279,A 0.000,B 0.000,C 90.000,E1 230.194} C_DIS
LIN {X 0.008,Y -152.180,Z 379.254,A 0.000,B 0.000,C 90.000,E1 225.688} C_DIS
LIN {X 0.024,Y -150.427,Z 379.239,A 0.000,B 0.000,C 90.000,E1 222.975} C_DIS
LIN {X -0.050,Y -147.155,Z 379.214,A 0.000,B 0.000,C 90.000,E1 218.463} C_DIS
LIN {X -0.083,Y -145.170,Z 379.193,A 0.000,B 0.000,C 90.000,E1 214.818} C_DIS
LIN {X -0.048,Y -142.320,Z 379.163,A 0.000,B 0.000,C 90.000,E1 209.283} C_DIS
LIN {X 0.073,Y -141.710,Z 379.152,A 0.000,B 0.000,C 90.000,E1 207.385} C_DIS
LIN {X -0.004,Y -139.471,Z 379.116,A 0.000,B 0.000,C 90.000,E1 200.918} C_DIS
LIN {X 0.050,Y -139.203,Z 379.106,A 0.000,B 0.000,C 90.000,E1 199.033} C_DIS
LIN {X -0.024,Y -138.329,Z 379.054,A 0.000,B 0.000,C 90.000,E1 189.726} C_DIS
LIN {X -0.021,Y -139.440,Z 379.007,A 0.000,B 0.000,C 90.000,E1 181.318} C_DIS
LIN {X 0.059,Y -140.974,Z 378.976,A 0.000,B 0.000,C 90.000,E1 175.698} C_DIS
LIN {X 0.009,Y -142.729,Z 378.956,A 0.000,B 0.000,C 90.000,E1 172.008} C_DIS
LIN {X -0.034,Y -145.115,Z 378.930,A 0.000,B 0.000,C 90.000,E1 167.409} C_DIS
LIN {X -0.040,Y -147.739,Z 378.910,A 0.000,B 0.000,C 90.000,E1 163.740} C_DIS
LIN {X 0.042,Y -150.403,Z 378.889,A 0.000,B 0.000,C 90.000,E1 160.061} C_DIS
LIN {X -0.083,Y -153.840,Z 378.869,A 0.000,B 0.000,C 90.000,E1 156.485} C_DIS
LIN {X -0.024,Y -157.251,Z 378.849,A 0.000,B 0.000,C 90.000,E1 152.871} C_DIS
LIN {X 0.054,Y -161.425,Z 378.829,A 0.000,B 0.000,C 90.000,E1 149.282} C_DIS
LIN {X -0.076,Y -165.626,Z 378.810,A 0.000,B 0.000,C 90.000,E1 145.801} C_DIS
LIN {X 0.044,Y -170.555,Z 378.790,A 0.000,B 0.000,C 90.000,E1 142.271} C_DIS
LIN {X -0.048,Y -175.434,Z 378.771,A 0.000,B 0.000,C 90.000,E1 138.852} C_DIS
LIN {X 0.069,Y -181.057,Z 378.752,A 0.000,B 0.000,C 90.000,E1 135.405} C_DIS
LIN {X -0.065,Y -186.494,Z 378.734,A 0.000,B 0.000,C 90.000,E1 132.081} C_DIS
LIN {X 0.003,Y -191.114,Z 378.720,A 0.000,B 0.000,C 90.000,E1 129.564} C_DIS
LIN {X -0.078,Y -196.909,Z 378.702,A 0.000,B 0.000,C 90.000,E1 126.297} C_DIS
LIN {X 0.015,Y -198.702,Z 378.696,A 0.000,B 0.000,C 90.000,E1 125.358} C_DIS
LIN {X -0.029,Y -298.776,Z 378.696,A 0.000,B 0.000,C 90.000,E1 125.358} C_DIS
LIN {X 0.056,Y -300.265,Z 378.696,A 0.000,B 0.000,C 90.000,E1 125.311} C_DIS
LIN {X 0.007,Y -303.965,Z 378.695,A 0.000,B 0.000,C 90.000,E1 125.152} C_DIS
LIN {X 0.032,Y -306.162,Z 378.694,A 0.000,B 0.000,C 90.000,E1 124.978} C_DIS
LIN {X 0.182,Y -309.222,Z 378.692,A 0.000,B 0.000,C 90.000,E1 124.612} C_DIS
LIN {X 0.087,Y -311.218,Z 378.691,A 0.000,B 0.000,C 90.000,E1 124.326} C_DIS
LIN {X -0.011,Y -312.784,Z 378.689,A 0.000,B 0.000,C 90.000,E1 124.040} C_DIS
LIN {X 0.039,Y -314.110,Z 378.687,A 0.000,B 0.000,C 90.000,E1 123.706} C_DIS
LIN {X -0.040,Y -325.469,Z 378.669,A 0.000,B 0.000,C 90.000,E1 120.512} C_DIS
LIN {X 0.188,Y -337.091,Z 378.654,A 0.000,B 0.000,C 90.000,E1 117.641} C_DIS
LIN {X -0.001,Y -350.166,Z 378.638,A 0.000,B 0.000,C 90.000,E1 114.899} C_DIS
LIN {X 0.149,Y -363.110,Z 378.625,A 0.000,B 0.000,C 90.000,E1 112.461} C_DIS
LIN {X 0.010,Y -377.391,Z 378.612,A 0.000,B 0.000,C 90.000,E1 110.120} C_DIS
LIN {X -0.039,Y -393.117,Z 378.599,A 0.000,B 0.000,C 90.000,E1 107.819} C_DIS
LIN {X 0.072,Y -410.403,Z 378.586,A 0.000,B 0.000,C 90.000,E1 105.552} C_DIS
LIN {X 0.115,Y -429.369,Z 378.574,A 0.000,B 0.000,C 90.000,E1 103.355} C_DIS
LIN {X 0.069,Y -449.482,Z 378.563,A 0.000,B 0.000,C 90.000,E1 101.299} C_DIS
LIN {X -0.142,Y -470.147,Z 378.552,A 0.000,B 0.000,C 90.000,E1 99.434} C_DIS
LIN {X 0.157,Y -488.640,Z 378.544,A 0.000,B 0.000,C 90.000,E1 97.871} C_DIS
LIN {X -0.164,Y -491.048,Z 378.543,A 0.000,B 0.000,C 90.000,E1 97.701} C_DIS
LIN {X 0.067,Y -492.876,Z 378.542,A 0.000,B 0.000,C 90.000,E1 97.466} C_DIS
LIN {X -0.095,Y -494.529,Z 378.540,A 0.000,B 0.000,C 90.000,E1 97.239} C_DIS
LIN {X -0.196,Y -495.766,Z 378.539,A 0.000,B 0.000,C 90.000,E1 97.004} C_DIS
LIN {X 0.055,Y -497.277,Z 378.536,A 0.000,B 0.000,C 90.000,E1 96.486} C_DIS
LIN {X -0.183,Y -497.724,Z 378.533,A 0.000,B 0.000,C 90.000,E1 96.024} C_DIS
LIN {X 0.035,Y -497.178,Z 378.531,A 0.000,B 0.000,C 90.000,E1 95.511} C_DIS
LIN {X -0.189,Y -495.548,Z 378.528,A 0.000,B 0.000,C 90.000,E1 95.049} C_DIS
LIN {X 0.211,Y -494.235,Z 378.527,A 0.000,B 0.000,C 90.000,E1 94.759} C_DIS
LIN {X -0.170,Y -488.916,Z 378.522,A 0.000,B 0.000,C 90.000,E1 94.069} C_DIS
LIN {X 0.214,Y -481.173,Z 378.517,A 0.000,B 0.000,C 90.000,E1 93.037} C_DIS
LIN {X -0.158,Y -457.670,Z 378.500,A 0.000,B 0.000,C 90.000,E1 90.057} C_DIS
LIN {X -0.104,Y -437.981,Z 378.484,A 0.000,B 0.000,C 90.000,E1 87.192} C_DIS
LIN {X -0.009,Y -418.482,Z 378.466,A 0.000,B 0.000,C 90.000,E1 83.970} C_DIS
LIN {X -0.018,Y -406.331,Z 378.454,A 0.000,B 0.000,C 90.000,E1 81.781} C_DIS
LIN {X -0.134,Y -394.459,Z 378.442,A 0.000,B 0.000,C 90.000,E1 79.567} C_DIS
LIN {X -0.180,Y -384.234,Z 378.431,A 0.000,B 0.000,C 90.000,E1 77.589} C_DIS
LIN {X -0.186,Y -371.148,Z 378.416,A 0.000,B 0.000,C 90.000,E1 74.991} C_DIS
LIN {X 0.047,Y -359.686,Z 378.403,A 0.000,B 0.000,C 90.000,E1 72.598} C_DIS
LIN {X 0.103,Y -348.425,Z 378.390,A 0.000,B 0.000,C 90.000,E1 70.188} C_DIS
LIN {X -0.203,Y -336.101,Z 378.375,A 0.000,B 0.000,C 90.000,E1 67.486} C_DIS
LIN {X -0.097,Y -321.895,Z 378.356,A 0.000,B 0.000,C 90.000,E1 64.024} C_DIS
LIN {X 0.102,Y -308.822,Z 378.336,A 0.000,B 0.000,C 90.000,E1 60.461} C_DIS
LIN {X 0.028,Y -297.758,Z 378.318,A 0.000,B 0.000,C 90.000,E1 57.199} C_DIS
LIN {X 0.035,Y -287.605,Z 378.299,A 0.000,B 0.000,C 90.000,E1 53.863} C_DIS
LIN {X -0.060,Y -280.079,Z 378.284,A 0.000,B 0.000,C 90.000,E1 51.170} C_DIS
LIN {X 0.021,Y -274.553,Z 378.273,A 0.000,B 0.000,C 90.000,E1 49.094} C_DIS
LIN {X -0.034,Y -268.896,Z 378.261,A 0.000,B 0.000,C 90.000,E1 47.025} C_DIS
LIN {X -0.021,Y -263.181,Z 378.250,A 0.000,B 0.000,C 90.000,E1 44.919} C_DIS
LIN {X 0.076,Y -257.393,Z 378.238,A 0.000,B 0.000,C 90.000,E1 42.771} C_DIS
LIN {X 0.077,Y -251.432,Z 378.226,A 0.000,B 0.000,C 90.000,E1 40.620} C_DIS
LIN {X 0.004,Y -243.388,Z 378.210,A 0.000,B 0.000,C 90.000,E1 37.729} C_DIS
LIN {X -0.037,Y -233.786,Z 378.189,A 0.000,B 0.000,C 90.000,E1 34.040} C_DIS
LIN {X 0.007,Y -224.713,Z 378.168,A 0.000,B 0.000,C 90.000,E1 30.256} C_DIS
LIN {X 0.037,Y -217.990,Z 378.151,A 0.000,B 0.000,C 90.000,E1 27.180} C_DIS
LIN {X 0.042,Y -210.477,Z 378.129,A 0.000,B 0.000,C 90.000,E1 23.281} C_DIS
LIN {X 0.040,Y -205.283,Z 378.112,A 0.000,B 0.000,C 90.000,E1 20.120} C_DIS
LIN {X -0.014,Y -199.610,Z 378.090,A 0.000,B 0.000,C 90.000,E1 16.134} C_DIS
LIN {X 0.060,Y -194.942,Z 378.067,A 0.000,B 0.000,C 90.000,E1 12.063} C_DIS
LIN {X -0.007,Y -191.270,Z 378.044,A 0.000,B 0.000,C 90.000,E1 7.992} C_DIS
LIN {X -0.070,Y -188.385,Z 378.012,A 0.000,B 0.000,C 90.000,E1 2.236} C_DIS
LIN {X 0.008,Y -189.578,Z 377.942,A 0.000,B 0.000,C 90.000,E1 349.577} C_DIS
LIN {X -0.002,Y -192.643,Z 377.915,A 0.000,B 0.000,C 90.000,E1 344.629} C_DIS
LIN {X -0.066,Y -196.321,Z 377.892,A 0.000,B 0.000,C 90.000,E1 340.550} C_DIS
LIN {X -0.058,Y -201.137,Z 377.869,A 0.000,B 0.000,C 90.000,E1 336.485} C_DIS
LIN {X -0.017,Y -205.745,Z 377.851,A 0.000,B 0.000,C 90.000,E1 333.256} C_DIS
LIN {X -0.025,Y -212.460,Z 377.829,A 0.000,B 0.000,C 90.000,E1 329.282} C_DIS
LIN {X -0.118,Y -219.685,Z 377.808,A 0.000,B 0.000,C 90.000,E1 325.388} C_DIS
LIN {X -0.016,Y -226.020,Z 377.790,A 0.000,B 0.000,C 90.000,E1 322.271} C_DIS
LIN {X -0.097,Y -234.740,Z 377.769,A 0.000,B 0.000,C 90.000,E1 318.485} C_DIS
LIN {X 0.077,Y -243.802,Z 377.751,A 0.000,B 0.000,C 90.000,E1 315.081} C_DIS
LIN {X 0.019,Y -252.813,Z 377.734,A 0.000,B 0.000,C 90.000,E1 312.162} C_DIS
LIN {X 0.044,Y -262.869,Z 377.718,A 0.000,B 0.000,C 90.000,E1 309.277} C_DIS
LIN {X 0.033,Y -273.462,Z 377.703,A 0.000,B 0.000,C 90.000,E1 306.457} C_DIS
LIN {X -0.082,Y -285.825,Z 377.685,A 0.000,B 0.000,C 90.000,E1 303.372} C_DIS
LIN {X -0.066,Y -301.279,Z 377.667,A 0.000,B 0.000,C 90.000,E1 300.001} C_DIS
LIN {X -0.063,Y -316.897,Z 377.650,A 0.000,B 0.000,C 90.000,E1 297.052} C_DIS
LIN {X -0.113,Y -330.599,Z 377.638,A 0.000,B 0.000,C 90.000,E1 294.823} C_DIS
LIN {X -0.122,Y -347.926,Z 377.624,A 0.000,B 0.000,C 90.000,E1 292.333} C_DIS
LIN {X 0.126,Y -363.650,Z 377.612,A 0.000,B 0.000,C 90.000,E1 290.174} C_DIS
LIN {X 0.046,Y -377.892,Z 377.602,A 0.000,B 0.000,C 90.000,E1 288.417} C_DIS
LIN {X 0.099,Y -403.564,Z 377.587,A 0.000,B 0.000,C 90.000,E1 285.607} C_DIS
LIN {X -0.021,Y -421.652,Z 377.577,A 0.000,B 0.000,C 90.000,E1 283.772} C_DIS
LIN {X 0.121,Y -431.812,Z 377.571,A 0.000,B 0.000,C 90.000,E1 282.715} C_DIS
LIN {X 0.112,Y -441.555,Z 377.565,A 0.000,B 0.000,C 90.000,E1 281.658} C_DIS
LIN {X 0.132,Y -450.396,Z 377.559,A 0.000,B 0.000,C 90.000,E1 280.602} C_DIS
LIN {X 0.171,Y -458.449,Z 377.553,A 0.000,B 0.000,C 90.000,E1 279.557} C_DIS
LIN {X -0.153,Y -465.677,Z 377.547,A 0.000,B 0.000,C 90.000,E1 278.568} C_DIS
LIN {X -0.003,Y -472.329,Z 377.542,A 0.000,B 0.000,C 90.000,E1 277.530} C_DIS
LIN {X -0.185,Y -478.330,Z 377.536,A 0.000,B 0.000,C 90.000,E1 276.543} C_DIS
LIN {X -0.227,Y -482.272,Z 377.532,A 0.000,B 0.000,C 90.000,E1 275.796} C_DIS
LIN {X -0.236,Y -485.575,Z 377.528,A 0.000,B 0.000,C 90.000,E1 275.049} C_DIS
LIN {X -0.046,Y -487.341,Z 377.525,A 0.000,B 0.000,C 90.000,E1 274.531} C_DIS
LIN {X 0.146,Y -488.713,Z 377.522,A 0.000,B 0.000,C 90.000,E1 274.012} C_DIS
LIN {X -0.171,Y -489.749,Z 377.520,A 0.000,B 0.000,C 90.000,E1 273.555} C_DIS
LIN {X 0.038,Y -490.485,Z 377.517,A 0.000,B 0.000,C 90.000,E1 273.037} C_DIS
LIN {X 0.226,Y -490.936,Z 377.514,A 0.000,B 0.000,C 90.000,E1 272.522} C_DIS
LIN {X -0.068,Y -491.077,Z 377.511,A 0.000,B 0.000,C 90.000,E1 272.064} C_DIS
LIN {X 0.147,Y -490.886,Z 377.509,A 0.000,B 0.000,C 90.000,E1 271.547} C_DIS
LIN {X -0.143,Y -490.348,Z 377.506,A 0.000,B 0.000,C 90.000,E1 271.088} C_DIS
LIN {X 0.057,Y -489.422,Z 377.503,A 0.000,B 0.000,C 90.000,E1 270.573} C_DIS
LIN {X -0.234,Y -488.017,Z 377.500,A 0.000,B 0.000,C 90.000,E1 270.115} C_DIS
LIN {X -0.042,Y -486.036,Z 377.498,A 0.000,B 0.000,C 90.000,E1 269.599} C_DIS
LIN {X -0.193,Y -484.862,Z 377.496,A 0.000,B 0.000,C 90.000,E1 269.370} C_DIS
LIN {X -0.020,Y -481.815,Z 377.494,A 0.000,B 0.000,C 90.000,E1 268.854} C_DIS
LIN {X 0.131,Y -477.868,Z 377.491,A 0.000,B 0.000,C 90.000,E1 268.339} C_DIS
LIN {X -0.021,Y -475.550,Z 377.489,A 0.000,B 0.000,C 90.000,E1 268.108} C_DIS
LIN {X 0.099,Y -469.759,Z 377.487,A 0.000,B 0.000,C 90.000,E1 267.593} C_DIS
LIN {X 0.189,Y -466.763,Z 377.485,A 0.000,B 0.000,C 90.000,E1 267.364} C_DIS
LIN {X 0.211,Y -460.079,Z 377.483,A 0.000,B 0.000,C 90.000,E1 266.963} C_DIS
LIN {X -0.061,Y -453.004,Z 377.481,A 0.000,B 0.000,C 90.000,E1 266.674} C_DIS
LIN {X 0.146,Y -445.821,Z 377.480,A 0.000,B 0.000,C 90.000,E1 266.388} C_DIS
LIN {X -0.135,Y -438.214,Z 377.479,A 0.000,B 0.000,C 90.000,E1 266.216} C_DIS
LIN {X -0.038,Y -430.032,Z 377.478,A 0.000,B 0.000,C 90.000,E1 266.045} C_DIS
LIN {X 0.005,Y -419.972,Z 377.477,A 0.000,B 0.000,C 90.000,E1 265.927} C_DIS
LIN {X 0.170,Y -410.554,Z 377.477,A 0.000,B 0.000,C 90.000,E1 265.869} C_DIS
LIN {X 0.039,Y -180.915,Z 377.477,A 0.000,B 0.000,C 90.000,E1 265.869} C_DIS
LIN {X 0.066,Y -180.824,Z 377.471,A 0.000,B 0.000,C 90.000,E1 264.837} C_DIS
LIN {X -0.039,Y -178.856,Z 377.442,A 0.000,B 0.000,C 90.000,E1 259.634} C_DIS
LIN {X 0.032,Y -175.900,Z 377.414,A 0.000,B 0.000,C 90.000,E1 254.519} C_DIS
LIN {X -0.029,Y -174.577,Z 377.405,A 0.000,B 0.000,C 90.000,E1 252.834} C_DIS
LIN {X 0.006,Y -171.561,Z 377.381,A 0.000,B 0.000,C 90.000,E1 248.539} C_DIS
LIN {X -0.011,Y -167.784,Z 377.357,A 0.000,B 0.000,C 90.000,E1 244.229} C_DIS
LIN {X 0.003,Y -166.498,Z 377.347,A 0.000,B 0.000,C 90.000,E1 242.487} C_DIS
LIN {X -0.002,Y -163.208,Z 377.328,A 0.000,B 0.000,C 90.000,E1 238.997} C_DIS
LIN {X -0.037,Y -161.172,Z 377.313,A 0.000,B 0.000,C 90.000,E1 236.373} C_DIS
LIN {X 0.088,Y -157.186,Z 377.289,A 0.000,B 0.000,C 90.000,E1 231.904} C_DIS
LIN {X 0.010,Y -155.916,Z 377.279,A 0.000,B 0.000,C 90.000,E1 230.150} C_DIS
LIN {X 0.067,Y -152.166,Z 377.254,A 0.000,B 0.000,C 90.000,E1 225.648} C_DIS
LIN {X -0.024,Y -150.415,Z 377.239,A 0.000,B 0.000,C 90.000,E1 222.975} C_DIS
LIN {X 0.017,Y -147.144,Z 377.213,A 0.000,B 0.000,C 90.000,E1 218.418} C_DIS
LIN {X 0.015,Y -145.702,Z 377.198,A 0.000,B 0.000,C 90.000,E1 215.678} C_DIS
LIN {X 0.022,Y -143.086,Z 377.173,A 0.000,B 0.000,C 90.000,E1 211.082} C_DIS
LIN {X 0.027,Y -141.703,Z 377.152,A 0.000,B 0.000,C 90.000,E1 207.385} C_DIS
LIN {X -0.050,Y -139.467,Z 377.116,A 0.000,B 0.000,C 90.000,E1 200.918} C_DIS
LIN {X 0.004,Y -139.200,Z 377.106,A 0.000,B 0.000,C 90.000,E1 199.033} C_DIS
LIN {X 0.067,Y -138.327,Z 377.054,A 0.000,B 0.000,C 90.000,E1 189.670} C_DIS
LIN {X -0.067,Y -139.444,Z 377.007,A 0.000,B 0.000,C 90.000,E1 181.318} C_DIS
LIN {X 0.013,Y -140.981,Z 376.976,A 0.000,B 0.000,C 90.000,E1 175.698} C_DIS
LIN {X -0.037,Y -142.737,Z 376.956,A 0.000,B 0.000,C 90.000,E1 172.008} C_DIS
LIN {X 0.061,Y -145.127,Z 376.930,A 0.000,B 0.000,C 90.000,E1 167.353} C_DIS
LIN {X 0.054,Y -147.750,Z 376.909,A 0.000,B 0.000,C 90.000,E1 163.685} C_DIS
LIN {X -0.006,Y -150.419,Z 376.889,A 0.000,B 0.000,C 90.000,E1 160.061} C_DIS
LIN {X 0.009,Y -153.859,Z 376.869,A 0.000,B 0.000,C 90.000,E1 156.433} C_DIS
LIN {X -0.074,Y -157.270,Z 376.849,A 0.000,B 0.000,C 90.000,E1 152.871} C_DIS
LIN {X 0.004,Y -161.448,Z 376.829,A 0.000,B 0.000,C 90.000,E1 149.282} C_DIS
LIN {X 0.010,Y -165.649,Z 376.810,A 0.000,B 0.000,C 90.000,E1 145.754} C_DIS
LIN {X -0.008,Y -170.583,Z 376.790,A 0.000,B 0.000,C 90.000,E1 142.271} C_DIS
LIN {X -0.101,Y -175.460,Z 376.771,A 0.000,B 0.000,C 90.000,E1 138.852} C_DIS
LIN {X 0.014,Y -181.083,Z 376.752,A 0.000,B 0.000,C 90.000,E1 135.405} C_DIS
LIN {X 0.005,Y -186.523,Z 376.734,A 0.000,B 0.000,C 90.000,E1 132.043} C_DIS
LIN {X -0.053,Y -191.141,Z 376.720,A 0.000,B 0.000,C 90.000,E1 129.564} C_DIS
LIN {X 0.025,Y -196.941,Z 376.701,A 0.000,B 0.000,C 90.000,E1 126.251} C_DIS
LIN {X 0.015,Y -198.796,Z 376.696,A 0.000,B 0.000,C 90.000,E1 125.311} C_DIS
LIN {X -0.030,Y -298.594,Z 376.696,A 0.000,B 0.000,C 90.000,E1 125.311} C_DIS
LIN {X -0.080,Y -303.550,Z 376.695,A 0.000,B 0.000,C 90.000,E1 125.152} C_DIS
LIN {X -0.057,Y -305.910,Z 376.694,A 0.000,B 0.000,C 90.000,E1 124.978} C_DIS
LIN {X 0.095,Y -309.100,Z 376.692,A 0.000,B 0.000,C 90.000,E1 124.612} C_DIS
LIN {X 0.049,Y -311.102,Z 376.691,A 0.000,B 0.000,C 90.000,E1 124.326} C_DIS
LIN {X 0.002,Y -312.678,Z 376.689,A 0.000,B 0.000,C 90.000,E1 124.040} C_DIS
LIN {X 0.052,Y -314.058,Z 376.687,A 0.000,B 0.000,C 90.000,E1 123.706} C_DIS
LIN {X -0.028,Y -325.439,Z 376.669,A 0.000,B 0.000,C 90.000,E1 120.512} C_DIS
LIN {X 0.200,Y -337.060,Z 376.654,A 0.000,B 0.000,C 90.000,E1 117.641} C_DIS
LIN {X 0.010,Y -350.134,Z 376.638,A 0.000,B 0.000,C 90.000,E1 114.899} C_DIS
LIN {X 0.159,Y -363.076,Z 376.625,A 0.000,B 0.000,C 90.000,E1 112.461} C_DIS
LIN {X 0.020,Y -377.357,Z 376.612,A 0.000,B 0.000,C 90.000,E1 110.120} C_DIS
LIN {X -0.030,Y -393.081,Z 376.599,A 0.000,B 0.000,C 90.000,E1 107.819} C_DIS
LIN {X 0.082,Y -410.365,Z 376.586,A 0.000,B 0.000,C 90.000,E1 105.552} C_DIS
LIN {X 0.124,Y -429.330,Z 376.574,A 0.000,B 0.000,C 90.000,E1 103.355} C_DIS
LIN {X 0.076,Y -449.442,Z 376.563,A 0.000,B 0.000,C 90.000,E1 101.299} C_DIS
LIN {X -0.136,Y -470.107,Z 376.552,A 0.000,B 0.000,C 90.000,E1 99.434} C_DIS
LIN {X -0.159,Y -491.055,Z 376.543,A 0.000,B 0.000,C 90.000,E1 97.701} C_DIS
LIN {X 0.071,Y -492.927,Z 376.542,A 0.000,B 0.000,C 90.000,E1 97.466} C_DIS
LIN {X -0.090,Y -494.616,Z 376.540,A 0.000,B 0.000,C 90.000,E1 97.239} C_DIS
LIN {X -0.191,Y -495.881,Z 376.539,A 0.000,B 0.000,C 90.000,E1 97.004} C_DIS
LIN {X 0.060,Y -497.435,Z 376.536,A 0.000,B 0.000,C 90.000,E1 96.486} C_DIS
LIN {X -0.177,Y -497.919,Z 376.533,A 0.000,B 0.000,C 90.000,E1 96.024} C_DIS
LIN {X 0.042,Y -497.409,Z 376.531,A 0.000,B 0.000,C 90.000,E1 95.511} C_DIS
LIN {X -0.181,Y -495.823,Z 376.528,A 0.000,B 0.000,C 90.000,E1 95.049} C_DIS
LIN {X 0.220,Y -494.536,Z 376.527,A 0.000,B 0.000,C 90.000,E1 94.759} C_DIS
LIN {X -0.159,Y -489.266,Z 376.522,A 0.000,B 0.000,C 90.000,E1 94.069} C_DIS
LIN {X 0.230,Y -481.527,Z 376.517,A 0.000,B 0.000,C 90.000,E1 93.037} C_DIS
LIN {X -0.133,Y -457.988,Z 376.500,A 0.000,B 0.000,C 90.000,E1 90.057} C_DIS
LIN {X -0.072,Y -438.259,Z 376.484,A 0.000,B 0.000,C 90.000,E1 87.192} C_DIS
LIN {X -0.113,Y -420.290,Z 376.468,A 0.000,B 0.000,C 90.000,E1 84.261} C_DIS
LIN {X 0.026,Y -406.596,Z 376.454,A 0.000,B 0.000,C 90.000,E1 81.781} C_DIS
LIN {X -0.085,Y -394.733,Z 376.442,A 0.000,B 0.000,C 90.000,E1 79.567} C_DIS
LIN {X -0.126,Y -384.526,Z 376.431,A 0.000,B 0.000,C 90.000,E1 77.589} C_DIS
LIN {X -0.127,Y -371.432,Z 376.417,A 0.000,B 0.000,C 90.000,E1 74.991} C_DIS
LIN {X 0.113,Y -359.948,Z 376.403,A 0.000,B 0.000,C 90.000,E1 72.598} C_DIS
LIN {X -0.156,Y -348.654,Z 376.390,A 0.000,B 0.000,C 90.000,E1 70.242} C_DIS
LIN {X -0.131,Y -336.295,Z 376.375,A 0.000,B 0.000,C 90.000,E1 67.486} C_DIS
LIN {X -0.022,Y -322.054,Z 376.356,A 0.000,B 0.000,C 90.000,E1 64.024} C_DIS
LIN {X 0.180,Y -308.983,Z 376.336,A 0.000,B 0.000,C 90.000,E1 60.461} C_DIS
LIN {X -0.143,Y -297.911,Z 376.318,A 0.000,B 0.000,C 90.000,E1 57.248} C_DIS
LIN {X -0.116,Y -287.768,Z 376.299,A 0.000,B 0.000,C 90.000,E1 53.909} C_DIS
LIN {X 0.023,Y -280.239,Z 376.284,A 0.000,B 0.000,C 90.000,E1 51.170} C_DIS
LIN {X 0.106,Y -274.717,Z 376.273,A 0.000,B 0.000,C 90.000,E1 49.094} C_DIS
LIN {X 0.051,Y -269.039,Z 376.261,A 0.000,B 0.000,C 90.000,E1 47.025} C_DIS
LIN {X 0.066,Y -263.330,Z 376.250,A 0.000,B 0.000,C 90.000,E1 44.919} C_DIS
LIN {X -0.025,Y -257.562,Z 376.238,A 0.000,B 0.000,C 90.000,E1 42.813} C_DIS
LIN {X -0.026,Y -251.610,Z 376.226,A 0.000,B 0.000,C 90.000,E1 40.663} C_DIS
LIN {X 0.083,Y -245.596,Z 376.214,A 0.000,B 0.000,C 90.000,E1 38.463} C_DIS
LIN {X -0.082,Y -235.871,Z 376.193,A 0.000,B 0.000,C 90.000,E1 34.818} C_DIS
LIN {X 0.002,Y -228.458,Z 376.177,A 0.000,B 0.000,C 90.000,E1 31.799} C_DIS
LIN {X 0.043,Y -219.752,Z 376.155,A 0.000,B 0.000,C 90.000,E1 27.975} C_DIS
LIN {X 0.092,Y -212.011,Z 376.134,A 0.000,B 0.000,C 90.000,E1 24.079} C_DIS
LIN {X -0.070,Y -206.597,Z 376.116,A 0.000,B 0.000,C 90.000,E1 20.972} C_DIS
LIN {X -0.079,Y -200.723,Z 376.094,A 0.000,B 0.000,C 90.000,E1 16.985} C_DIS
LIN {X 0.059,Y -196.700,Z 376.076,A 0.000,B 0.000,C 90.000,E1 13.716} C_DIS
LIN {X -0.035,Y -192.617,Z 376.054,A 0.000,B 0.000,C 90.000,E1 9.670} C_DIS
LIN {X -0.064,Y -189.764,Z 376.031,A 0.000,B 0.000,C 90.000,E1 5.568} C_DIS
LIN {X 0.063,Y -187.742,Z 375.993,A 0.000,B 0.000,C 90.000,E1 358.682} C_DIS
LIN {X 0.005,Y -189.510,Z 375.942,A 0.000,B 0.000,C 90.000,E1 349.577} C_DIS
LIN {X -0.008,Y -192.557,Z 375.915,A 0.000,B 0.000,C 90.000,E1 344.629} C_DIS
LIN {X -0.075,Y -196.251,Z 375.892,A 0.000,B 0.000,C 90.000,E1 340.550} C_DIS
LIN {X -0.069,Y -201.053,Z 375.869,A 0.000,B 0.000,C 90.000,E1 336.485} C_DIS
LIN {X -0.031,Y -205.667,Z 375.851,A 0.000,B 0.000,C 90.000,E1 333.256} C_DIS
LIN {X -0.041,Y -212.372,Z 375.829,A 0.000,B 0.000,C 90.000,E1 329.282} C_DIS
LIN {X 0.043,Y -219.565,Z 375.808,A 0.000,B 0.000,C 90.000,E1 325.341} C_DIS
LIN {X -0.040,Y -225.940,Z 375.790,A 0.000,B 0.000,C 90.000,E1 322.271} C_DIS
LIN {X 0.030,Y -234.657,Z 375.769,A 0.000,B 0.000,C 90.000,E1 318.447} C_DIS
LIN {X 0.046,Y -243.736,Z 375.751,A 0.000,B 0.000,C 90.000,E1 315.081} C_DIS
LIN {X -0.015,Y -252.743,Z 375.734,A 0.000,B 0.000,C 90.000,E1 312.162} C_DIS
LIN {X 0.007,Y -262.796,Z 375.718,A 0.000,B 0.000,C 90.000,E1 309.277} C_DIS
LIN {X 0.076,Y -274.742,Z 375.701,A 0.000,B 0.000,C 90.000,E1 306.091} C_DIS
LIN {X -0.126,Y -285.754,Z 375.685,A 0.000,B 0.000,C 90.000,E1 303.372} C_DIS
LIN {X -0.113,Y -301.279,Z 375.667,A 0.000,B 0.000,C 90.000,E1 300.001} C_DIS
LIN {X 0.169,Y -316.960,Z 375.650,A 0.000,B 0.000,C 90.000,E1 297.001} C_DIS
LIN {X 0.136,Y -330.759,Z 375.638,A 0.000,B 0.000,C 90.000,E1 294.771} C_DIS
LIN {X -0.172,Y -348.125,Z 375.624,A 0.000,B 0.000,C 90.000,E1 292.333} C_DIS
LIN {X 0.020,Y -361.583,Z 375.614,A 0.000,B 0.000,C 90.000,E1 290.482} C_DIS
LIN {X -0.127,Y -375.666,Z 375.604,A 0.000,B 0.000,C 90.000,E1 288.725} C_DIS
LIN {X 0.000,Y -401.123,Z 375.588,A 0.000,B 0.000,C 90.000,E1 285.898} C_DIS
LIN {X 0.172,Y -419.230,Z 375.578,A 0.000,B 0.000,C 90.000,E1 284.008} C_DIS
LIN {X -0.088,Y -429.427,Z 375.572,A 0.000,B 0.000,C 90.000,E1 283.008} C_DIS
LIN {X 0.143,Y -436.864,Z 375.568,A 0.000,B 0.000,C 90.000,E1 282.187} C_DIS
LIN {X -0.106,Y -443.920,Z 375.563,A 0.000,B 0.000,C 90.000,E1 281.422} C_DIS
LIN {X 0.134,Y -450.443,Z 375.559,A 0.000,B 0.000,C 90.000,E1 280.602} C_DIS
LIN {X -0.087,Y -456.522,Z 375.555,A 0.000,B 0.000,C 90.000,E1 279.849} C_DIS
LIN {X -0.190,Y -462.125,Z 375.550,A 0.000,B 0.000,C 90.000,E1 279.086} C_DIS
LIN {X -0.087,Y -469.037,Z 375.545,A 0.000,B 0.000,C 90.000,E1 278.049} C_DIS
LIN {X 0.108,Y -475.345,Z 375.539,A 0.000,B 0.000,C 90.000,E1 277.011} C_DIS
LIN {X 0.099,Y -479.652,Z 375.535,A 0.000,B 0.000,C 90.000,E1 276.258} C_DIS
LIN {X 0.070,Y -483.411,Z 375.531,A 0.000,B 0.000,C 90.000,E1 275.511} C_DIS
LIN {X -0.235,Y -485.546,Z 375.528,A 0.000,B 0.000,C 90.000,E1 275.049} C_DIS
LIN {X -0.047,Y -487.296,Z 375.525,A 0.000,B 0.000,C 90.000,E1 274.531} C_DIS
LIN {X 0.146,Y -488.650,Z 375.522,A 0.000,B 0.000,C 90.000,E1 274.012} C_DIS
LIN {X -0.172,Y -489.686,Z 375.520,A 0.000,B 0.000,C 90.000,E1 273.555} C_DIS
LIN {X 0.036,Y -490.402,Z 375.517,A 0.000,B 0.000,C 90.000,E1 273.037} C_DIS
LIN {X 0.225,Y -490.823,Z 375.514,A 0.000,B 0.000,C 90.000,E1 272.522} C_DIS
LIN {X -0.070,Y -490.962,Z 375.511,A 0.000,B 0.000,C 90.000,E1 272.064} C_DIS
LIN {X 0.144,Y -490.756,Z 375.509,A 0.000,B 0.000,C 90.000,E1 271.547} C_DIS
LIN {X -0.146,Y -490.265,Z 375.506,A 0.000,B 0.000,C 90.000,E1 271.088} C_DIS
LIN {X 0.053,Y -489.341,Z 375.503,A 0.000,B 0.000,C 90.000,E1 270.573} C_DIS
LIN {X -0.238,Y -487.943,Z 375.500,A 0.000,B 0.000,C 90.000,E1 270.115} C_DIS
LIN {X -0.046,Y -485.979,Z 375.498,A 0.000,B 0.000,C 90.000,E1 269.599} C_DIS
LIN {X -0.197,Y -484.810,Z 375.496,A 0.000,B 0.000,C 90.000,E1 269.370} C_DIS
LIN {X -0.025,Y -481.811,Z 375.494,A 0.000,B 0.000,C 90.000,E1 268.854} C_DIS
LIN {X -0.184,Y -479.995,Z 375.492,A 0.000,B 0.000,C 90.000,E1 268.625} C_DIS
LIN {X -0.026,Y -475.534,Z 375.489,A 0.000,B 0.000,C 90.000,E1 268.108} C_DIS
LIN {X -0.201,Y -472.897,Z 375.488,A 0.000,B 0.000,C 90.000,E1 267.879} C_DIS
LIN {X 0.094,Y -469.832,Z 375.487,A 0.000,B 0.000,C 90.000,E1 267.593} C_DIS
LIN {X 0.192,Y -466.853,Z 375.485,A 0.000,B 0.000,C 90.000,E1 267.364} C_DIS
LIN {X -0.176,Y -463.472,Z 375.484,A 0.000,B 0.000,C 90.000,E1 267.192} C_DIS
LIN {X 0.202,Y -460.241,Z 375.483,A 0.000,B 0.000,C 90.000,E1 266.963} C_DIS
LIN {X -0.087,Y -453.169,Z 375.481,A 0.000,B 0.000,C 90.000,E1 266.674} C_DIS
LIN {X 0.110,Y -445.957,Z 375.480,A 0.000,B 0.000,C 90.000,E1 266.388} C_DIS
LIN {X -0.184,Y -438.288,Z 375.479,A 0.000,B 0.000,C 90.000,E1 266.216} C_DIS
LIN {X -0.096,Y -429.975,Z 375.478,A 0.000,B 0.000,C 90.000,E1 266.045} C_DIS
LIN {X -0.055,Y -419.461,Z 375.477,A 0.000,B 0.000,C 90.000,E1 265.927} C_DIS
LIN {X 0.196,Y -415.283,Z 375.477,A 0.000,B 0.000,C 90.000,E1 265.869} C_DIS
LIN {X 0.050,Y -180.915,Z 375.477,A 0.000,B 0.000,C 90.000,E1 265.869} C_DIS
LIN {X 0.077,Y -180.825,Z 375.471,A 0.000,B 0.000,C 90.000,E1 264.837} C_DIS
LIN {X -0.030,Y -178.858,Z 375.442,A 0.000,B 0.000,C 90.000,E1 259.634} C_DIS
LIN {X 0.041,Y -175.901,Z 375.414,A 0.000,B 0.000,C 90.000,E1 254.519} C_DIS
LIN {X -0.020,Y -174.580,Z 375.405,A 0.000,B 0.000,C 90.000,E1 252.834} C_DIS
LIN {X 0.016,Y -171.563,Z 375.381,A 0.000,B 0.000,C 90.000,E1 248.539} C_DIS
LIN {X -0.003,Y -167.786,Z 375.357,A 0.000,B 0.000,C 90.000,E1 244.229} C_DIS
LIN {X 0.012,Y -166.501,Z 375.347,A 0.000,B 0.000,C 90.000,E1 242.487} C_DIS
LIN {X 0.008,Y -163.210,Z 375.328,A 0.000,B 0.000,C 90.000,E1 238.997} C_DIS
LIN {X -0.027,Y -161.175,Z 375.313,A 0.000,B 0.000,C 90.000,E1 236.373} C_DIS
LIN {X -0.028,Y -157.189,Z 375.289,A 0.000,B 0.000,C 90.000,E1 231.949} C_DIS
LIN {X 0.019,Y -155.918,Z 375.279,A 0.000,B 0.000,C 90.000,E1 230.150} C_DIS
LIN {X 0.075,Y -152.169,Z 375.254,A 0.000,B 0.000,C 90.000,E1 225.648} C_DIS
LIN {X -0.015,Y -150.418,Z 375.239,A 0.000,B 0.000,C 90.000,E1 222.975} C_DIS
LIN {X -0.089,Y -147.146,Z 375.214,A 0.000,B 0.000,C 90.000,E1 218.463} C_DIS
LIN {X 0.022,Y -145.704,Z 375.198,A 0.000,B 0.000,C 90.000,E1 215.678} C_DIS
LIN {X 0.030,Y -143.087,Z 375.173,A 0.000,B 0.000,C 90.000,E1 211.082} C_DIS
LIN {X 0.035,Y -141.704,Z 375.152,A 0.000,B 0.000,C 90.000,E1 207.385} C_DIS
LIN {X -0.042,Y -139.468,Z 375.116,A 0.000,B 0.000,C 90.000,E1 200.918} C_DIS
LIN {X 0.012,Y -139.201,Z 375.106,A 0.000,B 0.000,C 90.000,E1 199.033} C_DIS
LIN {X 0.075,Y -138.328,Z 375.054,A 0.000,B 0.000,C 90.000,E1 189.670} C_DIS
LIN {X -0.059,Y -139.444,Z 375.007,A 0.000,B 0.000,C 90.000,E1 181.318} C_DIS
LIN {X 0.020,Y -140.980,Z 374.976,A 0.000,B 0.000,C 90.000,E1 175.698} C_DIS
LIN {X -0.029,Y -142.736,Z 374.956,A 0.000,B 0.000,C 90.000,E1 172.008} C_DIS
LIN {X -0.072,Y -145.125,Z 374.930,A 0.000,B 0.000,C 90.000,E1 167.409} C_DIS
LIN {X 0.063,Y -147.749,Z 374.909,A 0.000,B 0.000,C 90.000,E1 163.685} C_DIS
LIN {X 0.002,Y -150.417,Z 374.889,A 0.000,B 0.000,C 90.000,E1 160.061} C_DIS
LIN {X 0.018,Y -153.857,Z 374.869,A 0.000,B 0.000,C 90.000,E1 156.433} C_DIS
LIN {X -0.065,Y -157.266,Z 374.849,A 0.000,B 0.000,C 90.000,E1 152.871} C_DIS
LIN {X 0.013,Y -161.444,Z 374.829,A 0.000,B 0.000,C 90.000,E1 149.282} C_DIS
LIN {X 0.019,Y -165.644,Z 374.810,A 0.000,B 0.000,C 90.000,E1 145.754} C_DIS
LIN {X 0.001,Y -170.578,Z 374.790,A 0.000,B 0.000,C 90.000,E1 142.271} C_DIS
LIN {X -0.091,Y -175.456,Z 374.771,A 0.000,B 0.000,C 90.000,E1 138.852} C_DIS
LIN {X 0.024,Y -181.078,Z 374.752,A 0.000,B 0.000,C 90.000,E1 135.405} C_DIS
LIN {X 0.015,Y -186.518,Z 374.734,A 0.000,B 0.000,C 90.000,E1 132.043} C_DIS
LIN {X -0.043,Y -191.136,Z 374.720,A 0.000,B 0.000,C 90.000,E1 129.564} C_DIS
LIN {X 0.035,Y -196.935,Z 374.701,A 0.000,B 0.000,C 90.000,E1 126.251} C_DIS
LIN {X 0.104,Y -198.906,Z 374.696,A 0.000,B 0.000,C 90.000,E1 125.231} C_DIS
LIN {X 0.106,Y -298.847,Z 374.696,A 0.000,B 0.000,C 90.000,E1 125.231} C_DIS
LIN {X -0.081,Y -303.596,Z 374.695,A 0.000,B 0.000,C 90.000,E1 125.105} C_DIS
LIN {X -0.043,Y -305.787,Z 374.694,A 0.000,B 0.000,C 90.000,E1 124.945} C_DIS
LIN {X 0.110,Y -308.804,Z 374.692,A 0.000,B 0.000,C 90.000,E1 124.612} C_DIS
LIN {X -0.042,Y -312.450,Z 374.689,A 0.000,B 0.000,C 90.000,E1 124.072} C_DIS
LIN {X 0.177,Y -313.917,Z 374.687,A 0.000,B 0.000,C 90.000,E1 123.706} C_DIS
LIN {X 0.019,Y -326.561,Z 374.668,A 0.000,B 0.000,C 90.000,E1 120.207} C_DIS
LIN {X -0.003,Y -338.324,Z 374.652,A 0.000,B 0.000,C 90.000,E1 117.385} C_DIS
LIN {X -0.168,Y -351.560,Z 374.637,A 0.000,B 0.000,C 90.000,E1 114.643} C_DIS
LIN {X 0.007,Y -364.654,Z 374.623,A 0.000,B 0.000,C 90.000,E1 112.206} C_DIS
LIN {X -0.105,Y -379.098,Z 374.610,A 0.000,B 0.000,C 90.000,E1 109.866} C_DIS
LIN {X 0.133,Y -394.998,Z 374.597,A 0.000,B 0.000,C 90.000,E1 107.528} C_DIS
LIN {X 0.019,Y -412.473,Z 374.585,A 0.000,B 0.000,C 90.000,E1 105.300} C_DIS
LIN {X 0.001,Y -431.641,Z 374.573,A 0.000,B 0.000,C 90.000,E1 103.119} C_DIS
LIN {X 0.023,Y -451.823,Z 374.562,A 0.000,B 0.000,C 90.000,E1 101.074} C_DIS
LIN {X -0.025,Y -472.547,Z 374.551,A 0.000,B 0.000,C 90.000,E1 99.208} C_DIS
LIN {X -0.050,Y -490.931,Z 374.543,A 0.000,B 0.000,C 90.000,E1 97.701} C_DIS
LIN {X 0.115,Y -492.879,Z 374.542,A 0.000,B 0.000,C 90.000,E1 97.473} C_DIS
LIN {X 0.018,Y -494.629,Z 374.540,A 0.000,B 0.000,C 90.000,E1 97.239} C_DIS
LIN {X -0.082,Y -495.941,Z 374.539,A 0.000,B 0.000,C 90.000,E1 97.004} C_DIS
LIN {X 0.169,Y -497.566,Z 374.536,A 0.000,B 0.000,C 90.000,E1 96.486} C_DIS
LIN {X -0.120,Y -498.110,Z 374.533,A 0.000,B 0.000,C 90.000,E1 96.030} C_DIS
LIN {X 0.152,Y -497.660,Z 374.531,A 0.000,B 0.000,C 90.000,E1 95.511} C_DIS
LIN {X -0.070,Y -496.143,Z 374.528,A 0.000,B 0.000,C 90.000,E1 95.049} C_DIS
LIN {X -0.204,Y -494.902,Z 374.527,A 0.000,B 0.000,C 90.000,E1 94.821} C_DIS
LIN {X -0.082,Y -489.682,Z 374.523,A 0.000,B 0.000,C 90.000,E1 94.073} C_DIS
LIN {X -0.136,Y -481.969,Z 374.517,A 0.000,B 0.000,C 90.000,E1 93.094} C_DIS
LIN {X 0.201,Y -460.281,Z 374.502,A 0.000,B 0.000,C 90.000,E1 90.286} C_DIS
LIN {X 0.138,Y -442.062,Z 374.487,A 0.000,B 0.000,C 90.000,E1 87.707} C_DIS
LIN {X 0.178,Y -423.790,Z 374.471,A 0.000,B 0.000,C 90.000,E1 84.780} C_DIS
LIN {X 0.114,Y -408.433,Z 374.456,A 0.000,B 0.000,C 90.000,E1 82.064} C_DIS
LIN {X 0.059,Y -395.085,Z 374.442,A 0.000,B 0.000,C 90.000,E1 79.567} C_DIS
LIN {X 0.022,Y -384.890,Z 374.431,A 0.000,B 0.000,C 90.000,E1 77.589} C_DIS
LIN {X 0.025,Y -371.770,Z 374.417,A 0.000,B 0.000,C 90.000,E1 74.991} C_DIS
LIN {X -0.144,Y -361.711,Z 374.405,A 0.000,B 0.000,C 90.000,E1 72.960} C_DIS
LIN {X -0.033,Y -350.354,Z 374.392,A 0.000,B 0.000,C 90.000,E1 70.550} C_DIS
LIN {X 0.028,Y -337.898,Z 374.377,A 0.000,B 0.000,C 90.000,E1 67.794} C_DIS
LIN {X 0.050,Y -323.525,Z 374.358,A 0.000,B 0.000,C 90.000,E1 64.357} C_DIS
LIN {X 0.015,Y -310.343,Z 374.338,A 0.000,B 0.000,C 90.000,E1 60.845} C_DIS
LIN {X 0.020,Y -298.117,Z 374.318,A 0.000,B 0.000,C 90.000,E1 57.248} C_DIS
LIN {X 0.048,Y -287.974,Z 374.300,A 0.000,B 0.000,C 90.000,E1 53.909} C_DIS
LIN {X -0.031,Y -280.441,Z 374.284,A 0.000,B 0.000,C 90.000,E1 51.215} C_DIS
LIN {X 0.063,Y -274.927,Z 374.273,A 0.000,B 0.000,C 90.000,E1 49.138} C_DIS
LIN {X -0.020,Y -267.335,Z 374.258,A 0.000,B 0.000,C 90.000,E1 46.377} C_DIS
LIN {X 0.062,Y -259.712,Z 374.242,A 0.000,B 0.000,C 90.000,E1 43.542} C_DIS
LIN {X 0.104,Y -253.862,Z 374.230,A 0.000,B 0.000,C 90.000,E1 41.391} C_DIS
LIN {X -0.096,Y -245.855,Z 374.214,A 0.000,B 0.000,C 90.000,E1 38.543} C_DIS
LIN {X 0.086,Y -236.105,Z 374.194,A 0.000,B 0.000,C 90.000,E1 34.818} C_DIS
